// TwinCAT 3 PLC project DemoApplication
// ProgramVersion: 3.1.4020.4
// libraries:
//   Tc2_PfwLib_Processing, * (Beckhoff Automation GmbH)
//   Tc2_Standard, * (Beckhoff Automation GmbH)
//   Tc2_System, * (Beckhoff Automation GmbH)
//   Tc2_Utilities, * (Beckhoff Automation GmbH)
//   Tc3_Interfaces, * (Beckhoff Automation GmbH)
//   Tc3_Module, * (Beckhoff Automation GmbH)
//   VisuDialogs, * (System)
// project tree:
//   DUTs/ E_HMIstatus.TcDUT, E_MainStateMachine.TcDUT, ST_TempLoad.TcDUT, ST_TempLoad_Cmd.TcDUT, ST_TempLoad_State.TcDUT, ST_TempSave.TcDUT, ST_TempSave_Cmd.TcDUT
//   GVLs/ GVL_10_Visu.TcGVL, GVL_20_Applikation.TcGVL, GVL_30_Scope.TcGVL
//   / PlcTask.TcTTO
//   POUs/ FB_Load.TcPOU, FB_MainVisu.TcPOU, FB_Save.TcPOU, MAIN.TcPOU
//   TextLists/ GlobalTextList.TcGTLO, TL_Params_BOOL.TcTLO, TL_Params_Enum.TcTLO, TL_Params_INT.TcTLO, TL_Mparams_LREAL.TcTLO, TL_TcPfw_ErrorId.TcTLO, TL_Pparmas.TcTLO, TL_Supply.TcTLO, TL_TctrlOutSelect.TcTLO, TL_TctrlPowerTerminal.TcTLO, TL_TempSensType.TcTLO, TL_TerminalType.TcTLO
//   VISUs/DUTs/ st_ParamsUnsave.TcDUT, ST_Param_Visu.TcDUT
//   VISUs/Pages/Load Save/ Visu_SaveLoad.TcVIS
//   VISUs/Pages/LoopTest/ Visu_LoopTest.TcVIS
//   VISUs/Pages/Machine/Parameter/ Param_BOOL.TcVIS, Param_DINT.TcVIS, Param_ENUM_PowerTerm.TcVIS, Param_ENUM_SelOut.TcVIS, Param_ENUM_SensType.TcVIS, Param_ENUM_TermType.TcVIS, Param_LREAL.TcVIS
//   VISUs/Pages/Machine/Subpage/ Visu_Mparam_Autotune.TcVIS, Visu_Mparam_Cool.TcVIS, Visu_Mparam_Extruder.TcVIS, Visu_Mparam_General.TcVIS, Visu_Mparam_Heat.TcVIS, Visu_Mparam_Supply.TcVIS, Visu_Mparam_Temperatur.TcVIS
//   VISUs/Pages/Machine/ Visu_MParam.TcVIS
//   VISUs/Pages/Product/ Param_LREAL_Pparam.TcVIS, Visu_PParam.TcVIS, Visu_PParam_Params.TcVIS
//   VISUs/Pages/Supply/ Param_LREAL_Supply.TcVIS, Visu_Supply.TcVIS, Visu_Supply_Params.TcVIS
//   VISUs/Pages/ Visu_Main.TcVIS
//   VISUs/POUs/ FB_Visu_Param.TcPOU, FB_Visu_Pparam.TcPOU, FB_Visu_Supply.TcPOU
//   VISUs/ VisualizationManager.TcVMO (not stored)
// real-time tasks:
//   TASK PlcTask: cycle T#1ms, priority 20, ADS port 350
//   TASK Task 3: cycle T#10ms, priority 1, ADS port 351
// I/O:
//   DEVICE Device 1 (EtherCAT) (disabled), AmsNetId 192.168.1.78.2.1
//     Term 1 (EK1100) [EK1100 EtherCAT Coupler (2A E-Bus)]
//       Term 2 (EL3314) [EL3314 4Ch. Ana. Input Thermocouple (TC)]
//       Term 3 (EL2889) [EL2889 16Ch. Dig. Output 24V, 0.5A, negative]
// variable links:
//   DemoApplication/DemoApplication Instance <-> Device 1 (EtherCAT)/Term 1 (EK1100)/Term 3 (EL2889)
//     PlcTask Outputs/.out_PfwTempCtrlOutput[1]/Htr_PwmPos <-> Channel 1/Output

CONFIGURATION DemoApplication
    RESOURCE PLC ON TwinCAT3
        TASK PlcTask(INTERVAL := T#1ms, PRIORITY := 20);
        PROGRAM MAIN WITH PlcTask : MAIN;
    END_RESOURCE
END_CONFIGURATION

// ---- DUTs/E_HMIstatus.TcDUT
TYPE E_HMIstatus :
(
	Off := 0,
	Standby,
	On,
	Autotune,
	IdleLoad
);
END_TYPE

// ---- DUTs/E_MainStateMachine.TcDUT
TYPE E_MainStateMachine :
(
	eMainSM_BasicInit := 0,
	eMainSM_TempInit,
	eMainSM_MParamLoad,
	eMainSM_PParamLoad,
	eMainSM_SupParamLoad,
	eMainSM_StartUp,
	eMainSM_Idle
);
END_TYPE

// ---- DUTs/ST_TempLoad.TcDUT
TYPE ST_TempLoad :
STRUCT
	stTempCmd: ST_TempLoad_Cmd;
	stTempState: ST_TempLoad_State;
END_STRUCT
END_TYPE

// ---- DUTs/ST_TempLoad_Cmd.TcDUT
TYPE ST_TempLoad_Cmd :
STRUCT
	bLoadPparams: BOOL;
	bLoadMparams: BOOL;
	bLoadSupplyParams: BOOL;
END_STRUCT
END_TYPE

// ---- DUTs/ST_TempLoad_State.TcDUT
TYPE ST_TempLoad_State :
STRUCT
	bPparamLoaded: BOOL;
	bMparamLoaded: BOOL;
	bPparamLoad: BOOL;
	bMparamLoad: BOOL;
	bSupplyParamsLoad: BOOL;
	bSupplyParamsLoaded: BOOL;
END_STRUCT
END_TYPE

// ---- DUTs/ST_TempSave.TcDUT
TYPE ST_TempSave :
STRUCT
	stTempCmd: ST_TempSave_Cmd;
END_STRUCT
END_TYPE

// ---- DUTs/ST_TempSave_Cmd.TcDUT
TYPE ST_TempSave_Cmd :
STRUCT
	bSavePparams: BOOL;
	bSaveMparams: BOOL;
	bSaveSupplyParams: BOOL;
END_STRUCT
END_TYPE

// ---- VISUs/DUTs/st_ParamsUnsave.TcDUT
TYPE st_ParamsUnsave :
STRUCT
	mParams:	ARRAY[cnPfwTempCtrlFirst..cnPfwTempCtrlLast] OF BOOL;
	pParams:	ARRAY[cnPfwTempCtrlFirst..cnPfwTempCtrlLast] OF BOOL;
	supply:		ARRAY[cnPfwAppSupplyFirst..cnPfwAppSupplyLast] OF BOOL;
END_STRUCT
END_TYPE

// ---- VISUs/DUTs/ST_Param_Visu.TcDUT
TYPE ST_Param_Visu :
STRUCT
	 nActiveParamList: INT:=0;
	 
	sInUse:				STRING;
	 
	 bBoolAktValue:		ARRAY[1..cnParamsArrayLast] OF BOOL;
	 bBoolNewValue:		ARRAY[1..cnParamsArrayLast] OF BOOL;
	 bBoolSetValue:		ARRAY[1..cnParamsArrayLast] OF BOOL;

	 fLrealAktValue:	ARRAY[1..cnParamsArrayLast] OF LREAL;
	 fLrealNewValue:	ARRAY[1..cnParamsArrayLast] OF LREAL;
	 bLrealSetValue:	ARRAY[1..cnParamsArrayLast] OF BOOL;
	 
	 nDintAktValue:		ARRAY[1..cnParamsArrayLast] OF DINT;
	 nDintNewValue:		ARRAY[1..cnParamsArrayLast] OF DINT;
	 bDintSetValue:		ARRAY[1..cnParamsArrayLast] OF BOOL;
	 
	 nEnumAktValue:		ARRAY[1..cnParamsArrayLast] OF DINT;
	 nEnumNewValue:		ARRAY[1..cnParamsArrayLast] OF DINT;
	 bEnumSetValue:		ARRAY[1..cnParamsArrayLast] OF BOOL;
	 	 
END_STRUCT
END_TYPE

// ---- GVLs/GVL_10_Visu.TcGVL
VAR_GLOBAL CONSTANT
	cnParamsArrayLast:				INT:=50;
END_VAR

VAR_GLOBAL
	nVisuCount: INT:=cnPfwTempCtrlFirst;
	nSupplyCnt:	INT:=cnPfwAppSupplyFirst;
	
	eStatus: E_HMIstatus:=Off;
	
	bVisuNext: BOOL;
	bVisuBefore: BOOL;
	
	bVisuAutotune: BOOL;
	bVisuIdleLoad: BOOL;
	bVisuIdleLoadAktiv: BOOL;
	
	bGlobalError: BOOL;
	
	bParamsInit: BOOL:=FALSE;
	
	sErrorText:	STRING;
	
	
	
	
	stMParam_Visu:	ST_Param_Visu;
	stPParam_Visu:	ST_Param_Visu;
	stSupply_Visu:	ST_Param_Visu;
	stParamsUnsave:	st_ParamsUnsave;
	

	GlobalOne:INT:=1;
		A:INT:=0;
END_VAR

// ---- GVLs/GVL_20_Applikation.TcGVL
VAR_GLOBAL

	stTempLoad: ST_TempLoad;
	stTempSave: ST_TempSave;
	
END_VAR

// ---- GVLs/GVL_30_Scope.TcGVL
VAR_GLOBAL
	Scope_TempCtrlVariables: FB_Scope_TempCtrlVariables;
END_VAR

// ---- POUs/MAIN.TcPOU
PROGRAM MAIN
VAR
	eState: E_MainStateMachine := eMainSM_BasicInit;
	nCount: INT := 0;
	fCycleTime: LREAL := 0.025;
	fbTempCtrl: FB_TempCtrlMainBody_TcPfw_TC3;
	fbVisu: FB_MainVisu;

	bEntry:	BOOL;
	fbSave: FB_Save;
	fbLoad: FB_Load;
END_VAR


CASE eState OF
	eMainSM_BasicInit:
		_01_BasicInit();
		bEntry:=TRUE;
		eState:=eMainSM_MParamLoad;
		
	eMainSM_TempInit:
		_02_ParamsInit();
		bParamsInit:=FALSE;
		eState:=eMainSM_Idle;
		
	eMainSM_MParamLoad:
		IF bEntry THEN
			bEntry:=FALSE;
			stTempLoad.stTempCmd.bLoadMparams:=TRUE;
		ELSE
			IF stTempLoad.stTempState.bMparamLoaded THEN
				eState:=eMainSM_PParamLoad;
				bEntry:=TRUE;
			END_IF
		END_IF

		
	eMainSM_PParamLoad:
		IF bEntry THEN
			bEntry:=FALSE;
			stTempLoad.stTempCmd.bLoadPparams:=TRUE;
		ELSE
			IF stTempLoad.stTempState.bPparamLoaded THEN
				eState:=eMainSM_SupParamLoad;
				bEntry:=TRUE;
			END_IF
		END_IF

		
	eMainSM_SupParamLoad:
		IF bEntry THEN
			bEntry:=FALSE;
			stTempLoad.stTempCmd.bLoadSupplyParams:=TRUE;
		ELSE
			IF stTempLoad.stTempState.bSupplyParamsLoaded THEN
				eState:=eMainSM_StartUp;
				bEntry:=TRUE;
			END_IF
		END_IF

		
	eMainSM_StartUp:
		bEntry:=FALSE;
		fbTempCtrl.ConfigEnable:=TRUE;
		(*
		fbTempCtrl.tCycle:=fCycleTime;
		*)
		fbTempCtrl.tCycle:=0.025;
		fbTempCtrl.Looptest_Enable:=FALSE;
		fbTempCtrl.Callback_Enable:=TRUE;
		fbTempCtrl.Simu_Enable:=TRUE;
		eState:=eMainSM_Idle;
	
	eMainSM_Idle:
		IF bParamsInit THEN
			eState:=eMainSM_TempInit;
		END_IF
		
END_CASE

fbTempCtrl(
	Looptest_Enable:= TRUE,
	Scope_TempCtrlVariables:=Scope_TempCtrlVariables);
	
fbVisu();

fbSave();
fbLoad();

ACTION _01_BasicInit:
// Get Cycle Time
IF(GETCURTASKINDEXEX()<=0)THEN
	fCycletime:=0.025;		(* don't know, just guessing *)
ELSE
	fCycletime:=UDINT_TO_LREAL(_TaskInfo[GETCURTASKINDEXEX()].cycleTime)/10000000.0;
END_IF

// Init Zone ID/Name
FOR nCount := cnPfwTempCtrlFirst TO cnPfwTempCtrlLast DO
	aaaPfwTempMparamFromHmi[nCount].ZoneId := nCount;				(* zone id	*)
	aaaPfwTempMparamFromHmi[nCount].ZoneName := CONCAT('Zone_', INT_TO_STRING(nCount));	(* zonen name	*)
END_FOR
END_ACTION

ACTION _02_ParamsInit:
(* initialize of the machine parameter*)
	FOR nCount := cnPfwTempCtrlFirst TO cnPfwTempCtrlLast DO
		aaaPfwTempMparamFromHmi[nCount].AbsoluteHigh:=300;											(* limiting value of absolut hight.	*)
		aaaPfwTempMparamFromHmi[nCount].AbsoluteLow:=100;											(* limiting value of absolut low.	*)
		aaaPfwTempMparamFromHmi[nCount].InUse:=TRUE;												(* Zone is in use	*)
		aaaPfwTempMparamFromHmi[nCount].Enable:=TRUE;
		aaaPfwTempMparamFromHmi[nCount].SensorType:=0;												(* simulation	*)
		aaaPfwTempMparamFromHmi[nCount].ExtruderId:=1;												(* simulation	*)
		aaaPfwTempMparamFromHmi[nCount].TempSensTerm:=0;											(* simulation	*)
		aaaPfwTempMparamFromHmi[nCount].ZoneId:=nCount;												(* zone id		*)
		aaaPfwTempMparamFromHmi[nCount].ZoneName:=CONCAT('Zone_', INT_TO_STRING(nCount));(* zone name	*)
		IF(aaaPfwTempMparamFromHmi[nCount].KpCool<0.1)THEN
			aaaPfwTempMparamFromHmi[nCount].KpCool:=0.1;													(* default Kp cooling	*)
		END_IF
		IF(aaaPfwTempMparamFromHmi[nCount].KpHeat<0.1)THEN
			aaaPfwTempMparamFromHmi[nCount].KpHeat:=0.2;													(* default Kp heating 	*)
		END_IF
(*		aaaPfwTempMparamFromHmi[nCount].SettlingTime:=5.0;											(* Settling Time	*)*)
//		aaaPfwTempMparamFromHmi[nCount].SupplyLoad_Cooler:=100; 									(* coolingpower	*)
		aaaPfwTempMparamFromHmi[nCount].SupplyLoad_Heater:=1200;	 								(* heatingpower	*)
		aaaPfwTempMparamFromHmi[nCount].TuneEnd:=80;													(* Tune End % of setpoint	*)
		aaaPfwTempMparamFromHmi[nCount].TuneKp:=1.2;													(* Kp Tuning	*)
		aaaPfwTempMparamFromHmi[nCount].TuneTd:=0.25;												(* Td Tuning	*)
		aaaPfwTempMparamFromHmi[nCount].TuneTn:=2;													(* Tn Tuning	*)
		aaaPfwTempMparamFromHmi[nCount].TuneTv:=0.5;													(* Tv Tuning	*)
		aaaPfwTempMparamFromHmi[nCount].TuneY:=100;													(* Y Tuning		*)
		aaaPfwTempMparamFromHmi[nCount].Ramping_Rate:=0.005;										(* ramping rate	*)
		aaaPfwTempMparamFromHmi[nCount].Ramping_Tolerance:= 10;									(*	ramping tolerance*)
		aaaPfwTempMparamFromHmi[nCount].OutputSel_H:=eTcPfwTcOut_PWM;							(*	Heating output signal	*)
		aaaPfwTempMparamFromHmi[nCount].OutputSel_C:=eTcPfwTcOut_NoSignal;							(*	cooling output signal	*)
		aaaPfwTempMparamFromHmi[nCount].UseCooling:=FALSE;											(* cooling on	*)
		aaaPfwTempMparamFromHmi[nCount].TuneCooling:=FALSE;											(* cooling on	*)
		aaaPfwTempMparamFromHmi[nCount].ExtruderCompEna:=FALSE;											(* extruder comp	*)
		aaaPfwTempMparamFromHmi[nCount].fc_Enable:=FALSE;											(* Zwangskuelung	*)
		aaaPfwTempMparamFromHmi[nCount].fc_OffTime:=600.0;											(* Zwangskuelung	*)
		aaaPfwTempMparamFromHmi[nCount].fc_OnTime:=10.0;											(* Zwangskuelung	*)

(*		aaaPfwTempMparamFromHmi[nCount].SupplyLoad_Tolerance:=20.0;											(* Supply Tolerance	*)*)

		aaaPfwTempMparamFromHmi[nCount].SupplyLoad_Tolerance:=0.0;											(* Supply Tolerance	*)

		aaaPfwTempMparamFromHmi[nCount].SupplyId:=1;
		aaaPfwTempMparamFromHmi[nCount].ModuleId:=1;
	END_FOR
	(* mapping of the zones to the module and supply lines	*)


	(* initialize of the product parameter*)
	FOR nCount := cnPfwTempCtrlFirst TO cnPfwTempCtrlLast DO
		aaaPfwTempPparamFromHmi[nCount].Setpoint:=180;
		aaaPfwTempPparamFromHmi[nCount].StandbySetpoint:=18;
		aaaPfwTempPparamFromHmi[nCount].Threshold_M:=-10;
		aaaPfwTempPparamFromHmi[nCount].Threshold_MM:=-15;
		aaaPfwTempPparamFromHmi[nCount].Threshold_P:=10;
		aaaPfwTempPparamFromHmi[nCount].Threshold_PP:=15;
		aaaPfwTempPparamFromHmi[nCount].Update:=TRUE;
	END_FOR

	(* initialize of the supply lines*)
	FOR nCount := cnPfwAppSupplyFirst TO cnPfwAppSupplyLast DO
		stPfwSupplyLineCfg[nCount].fPwmCycleTime:=1;
		stPfwSupplyLineCfg[nCount].fPwmMaxOnTime:=1.0;
		stPfwSupplyLineCfg[nCount].fPwmMinOnTime:=0.1;
		stPfwSupplyLineCfg[nCount].fPwmMaxRampLoad:=1;
		stPfwSupplyLineCfg[nCount].nPwmFactorC:=10;
	END_FOR
END_ACTION

END_PROGRAM

// ---- POUs/FB_MainVisu.TcPOU
FUNCTION_BLOCK FB_MainVisu
VAR
	bOldVisuNext: BOOL;
	ncount: INT;
	bAutotuneAllDone: BOOL;
	eOldState: E_HMIstatus;
	bEntry:		BOOL:=TRUE;
	
	nIdx:				INT;
	fbVisuMParam:		FB_Visu_Param;
	fbVisuPParam:		FB_Visu_PParam;
	fbVisuSupply:		FB_Visu_Supply;
	(*
	fbVisu_Mparam:		FB_Visu_Mparam;
	fbVisu_Pparam:		FB_Visu_Pparam;
	fbVisu_Supply:		FB_Visu_Supply;
	*)
END_VAR

//
//		All Zones
//

bEntry:=(eStatus<>eOldState);
eOldState:=eStatus;

CASE eStatus OF

	Off:
		IF bEntry THEN
			FOR ncount:=cnPfwTempCtrlFirst TO cnPfwTempCtrlLast DO
				aaaPfwTempMparamFromHmi[ncount].Enable:=FALSE;
				stPfwTempCtrl[nCount].Enable:=FALSE;
			END_FOR
			bEntry:=FALSE;
		END_IF
	
	Standby:
		IF bEntry THEN
			FOR ncount:=cnPfwTempCtrlFirst TO cnPfwTempCtrlLast DO
				IF aaaPfwTempToHmi[nCount].InUse THEN
					stPfwTempCtrl[nCount].SelSetpoint:=TRUE;
					aaaPfwTempMparamFromHmi[ncount].Enable:=TRUE;
					stPfwTempCtrl[nCount].Enable:=TRUE;
				END_IF
			END_FOR
			bEntry:=FALSE;
		END_IF
	
	On:
		IF bEntry THEN
			FOR ncount:=cnPfwTempCtrlFirst TO cnPfwTempCtrlLast DO
				IF aaaPfwTempToHmi[nCount].InUse THEN
					stPfwTempCtrl[nCount].SelSetpoint:=FALSE;
					aaaPfwTempMparamFromHmi[ncount].Enable:=TRUE;
					stPfwTempCtrl[nCount].Enable:=TRUE;
				END_IF
			END_FOR
			bEntry:=FALSE;
		END_IF
	
	Autotune:
		IF bEntry THEN
			FOR ncount:=cnPfwTempCtrlFirst TO cnPfwTempCtrlLast DO
				IF aaaPfwTempToHmi[nCount].InUse THEN
					stPfwTempCtrl[nCount].Enable:=TRUE;
					aaaPfwTempMparamFromHmi[ncount].Enable:=TRUE;
					aaaPfwTempMparamFromHmi[ncount].Autotune:=TRUE;
				END_IF
			END_FOR
		ELSE
			bAutotuneAllDone:=TRUE;
			FOR ncount:=cnPfwTempCtrlFirst TO cnPfwTempCtrlLast DO
				IF(aaaPfwTempToHmi[nCount].TuningDone OR aaaPfwTempToHmi[nCount].Error) THEN
					IF aaaPfwTempToHmi[nCount].InUse THEN
						stPfwTempCtrl[nCount].Enable:=FALSE;
						aaaPfwTempMparamFromHmi[ncount].Enable:=FALSE;
						aaaPfwTempMparamFromHmi[ncount].Autotune:=FALSE;
					END_IF
				ELSE
					bAutoTuneAllDone:=FALSE;
				END_IF
			END_FOR
			IF bAutotuneAllDone THEN
				eStatus:=Standby;
			END_IF
		END_IF
		
	IdleLoad:
		IF bEntry THEN
			FOR ncount:=cnPfwTempCtrlFirst TO cnPfwTempCtrlLast DO
				IF aaaPfwTempToHmi[ncount].Enable THEN
					aaaPfwTempMparamFromHmi[ncount].Ena_TuneIdleLoad:=TRUE;
				END_IF
			END_FOR
		ELSE
			FOR ncount:=cnPfwTempCtrlFirst TO cnPfwTempCtrlLast DO
				bVisuIdleLoadAktiv:=FALSE;
				IF(aaaPfwTempToHmi[ncount].IdleLoadActive)THEN
					bVisuIdleLoadAktiv:=TRUE;
				END_IF
			END_FOR
			IF NOT bVisuIdleLoadAktiv THEN
				eStatus:=On;
			END_IF
		END_IF
END_CASE



//
//		Selected Zone
//

// Select Zone
IF(bVisuNext)THEN
	nVisuCount:=MIN(nVisuCount+1,cnPfwTempCtrlLast);
	bVisuNext:=FALSE;
ELSIF(bVisuBefore)THEN
	nVisuCount:=MAX(nVisuCount-1,cnPfwTempCtrlFirst);
	bVisuBefore:=FALSE;
END_IF

IF(bVisuAutotune)THEN
	aaaPfwTempMparamFromHmi[nVisuCount].Autotune:=TRUE;
ELSIF bVisuIdleLoad THEN
	aaaPfwTempMparamFromHmi[nVisuCount].Ena_TuneIdleLoad:=TRUE;
END_IF



ErrorHandling();
fbVisuMParam(stMParam_Visu:=stMParam_Visu, stParamsUnsave:=stParamsUnsave);
fbVisuPParam(stPParam_Visu:=stPParam_Visu, stParamsUnsave:=stParamsUnsave);
fbVisuSupply(stSupply_Visu:=stSupply_Visu, stParamsUnsave:=stParamsUnsave);

ACTION ErrorHandling:
bGlobalError:=FALSE;
sErrorText:='No Error';
FOR ncount:=cnPfwTempCtrlFirst TO cnPfwTempCtrlLast DO
	IF aaaPfwTempToHmi[ncount].Error THEN
		IF sErrorText='No Error' THEN
			sErrorText:='Error in Zone ';
		ELSE
			sErrorText:=CONCAT(sErrorText, ', ');
		END_IF
		sErrorText:=CONCAT(sErrorText, INT_TO_STRING(ncount));
		bGlobalError:=TRUE;
	END_IF
END_FOR
END_ACTION

END_FUNCTION_BLOCK

// ---- VISUs/POUs/FB_Visu_Param.TcPOU
FUNCTION_BLOCK FB_Visu_Param
VAR_IN_OUT
	stMParam_Visu:	ST_Param_Visu;
	stParamsUnsave:st_ParamsUnsave;
END_VAR
VAR
	nIdx:INT;
END_VAR

IF aaaPfwTempMparamFromHmi[nVisuCount].InUse THEN
	stMParam_Visu.sInUse:='Is In Use';
ELSE
	stMParam_Visu.sInUse:='Not In Use'; 
END_IF




FOR nIdx:=1 TO cnParamsArrayLast BY 1 DO
	// Get
	stMParam_Visu.bBoolAktValue[nIdx]:=GetBOOL(nVisuCount, nIdx);
	stMParam_Visu.fLrealAktValue[nIdx]:=GetLreal(nVisuCount, nIdx);
	stMParam_Visu.nDintAktValue[nIdx]:=GetInt(nVisuCount, nIdx);
	stMParam_Visu.nEnumAktValue[nIdx]:=GetEnum(nVisuCount, nIdx);
	
	// Set
	IF stMParam_Visu.bBoolSetValue[nIdx] THEN
		stMParam_Visu.bBoolSetValue[nIdx]:=FALSE;
		SetBool(nVisuCount,nIdx);
	END_IF
	
	IF stMParam_Visu.bLrealSetValue[nIdx] THEN
		stMParam_Visu.bLrealSetValue[nIdx]:=FALSE;
		SetLreal(nVisuCount,nIdx, stMParam_Visu.fLrealNewValue[nidx]);
	END_IF
	
	
	IF stMParam_Visu.bDintSetValue[nIdx] THEN
		stMParam_Visu.bDintSetValue[nIdx]:=FALSE;
		SetInt(nVisuCount,nIdx,DINT_TO_INT(stMParam_Visu.nDintNewValue[nidx]));
	END_IF
	
	IF stMParam_Visu.bEnumSetValue[nIdx] THEN
		stMParam_Visu.bEnumSetValue[nIdx]:=FALSE;
		SetEnum(nVisuCount,nIdx,stMParam_Visu.nEnumNewValue[nidx]);
	END_IF
END_FOR

METHOD SetInt : INT
VAR_INPUT
	nZone:	INT;
	nIdx:	INT;
	nValue:	INT;
END_VAR
CASE nIdx OF 
1:
	aaaPfwTempMparamFromHmi[nZone].App_HmiType:=nValue;
2:
	aaaPfwTempMparamFromHmi[nZone].TermChannel:=nValue;
3:
	aaaPfwTempMparamFromHmi[nZone].ExtruderId:=nValue;
4:
	aaaPfwTempMparamFromHmi[nZone].ModuleId:=nValue;
5:
	aaaPfwTempMparamFromHmi[nZone].ZoneId:=nValue;
6:
	aaaPfwTempMparamFromHmi[nZone].SupplyId:=nValue;
7:
	aaaPfwTempMparamFromHmi[nZone].CJ_CompMode:=nValue;
8:
	aaaPfwTempMparamFromHmi[nZone].CJ_CompZone:=nValue;
9:
	aaaPfwTempMparamFromHmi[nZone].SensTermSwapIdx:=nValue;
10:
	aaaPfwTempMparamFromHmi[nZone].HeaterSwapIdx:=nValue;
11:
	aaaPfwTempMparamFromHmi[nZone].CoolerSwapIdx:=nValue;
12:
	aaaPfwTempMparamFromHmi[nZone].nPwmFactorC:=nValue;

ELSE
	;
END_CASE

stParamsUnsave.mParams[nZone]:=TRUE;
END_METHOD

METHOD SetEnum : DINT
VAR_INPUT
	nZone:	INT;
	nIdx:	INT;
	nValue:	DINT;
END_VAR
CASE nIdx OF 

1:
	aaaPfwTempMparamFromHmi[nZone].OutputSel_H:=DINT_TO_INT(nValue);
2:
	aaaPfwTempMparamFromHmi[nZone].OutputSel_C:=DINT_TO_INT(nValue);
3:
	aaaPfwTempMparamFromHmi[nZone].TempSensTerm:=DINT_TO_INT(nValue);
4:
	aaaPfwTempMparamFromHmi[nZone].SensorType:=DINT_TO_INT(nValue);
ELSE
;
END_CASE
	
stParamsUnsave.mParams[nZone]:=TRUE;
END_METHOD

METHOD GetEnum : DINT
VAR_INPUT
	nZone:	INT;
	nIdx:	INT;
END_VAR
CASE nIdx OF 

1:
	GetEnum:=aaaPfwTempMparamFromHmi[nZone].OutputSel_H;
2:
	GetEnum:=aaaPfwTempMparamFromHmi[nZone].OutputSel_C;
3:
	GetEnum:=aaaPfwTempMparamFromHmi[nZone].TempSensTerm;
4:
	GetEnum:=aaaPfwTempMparamFromHmi[nZone].SensorType;
ELSE
	GetEnum:=-1;
END_CASE
END_METHOD

METHOD GetLreal : LREAL
VAR_INPUT
	nZone:	INT;
	nIdx:	INT;
END_VAR
VAR
END_VAR
CASE nIdx OF 
1:
	GetLreal:=aaaPfwTempMparamFromHmi[nZone].AbsoluteHigh;
2:
	GetLreal:=aaaPfwTempMparamFromHmi[nZone].AbsoluteLow;
3:
	GetLreal:=aaaPfwTempMparamFromHmi[nZone].ExtruderComp;
4:
	GetLreal:=aaaPfwTempMparamFromHmi[nZone].KpCool;
5:
	GetLreal:=aaaPfwTempMparamFromHmi[nZone].KpHeat;
6:
	GetLreal:=aaaPfwTempMparamFromHmi[nZone].TdCool;
7:
	GetLreal:=aaaPfwTempMparamFromHmi[nZone].TdHeat;
8:
	GetLreal:=aaaPfwTempMparamFromHmi[nZone].TnCool;
9:
	GetLreal:=aaaPfwTempMparamFromHmi[nZone].TnHeat;
10:
	GetLreal:=aaaPfwTempMparamFromHmi[nZone].TvCool;
11:
	GetLreal:=aaaPfwTempMparamFromHmi[nZone].TvHeat;
12:
	GetLreal:=aaaPfwTempMparamFromHmi[nZone].Overshoot;
13:
	GetLreal:=aaaPfwTempMparamFromHmi[nZone].Tracking_Rate;
14:
	GetLreal:=aaaPfwTempMparamFromHmi[nZone].Tracking_Td;
15:
	GetLreal:=aaaPfwTempMparamFromHmi[nZone].Ramping_Rate;
16:
	GetLreal:=aaaPfwTempMparamFromHmi[nZone].Ramping_RateC;
17:
	GetLreal:=aaaPfwTempMparamFromHmi[nZone].Ramping_Tolerance;
18:
	GetLreal:=aaaPfwTempMparamFromHmi[nZone].dTmax;
19:
	GetLreal:=aaaPfwTempMparamFromHmi[nZone].SensorOffset;
20:
	GetLreal:=aaaPfwTempMparamFromHmi[nZone].SettlingTime;
21:
	GetLreal:=aaaPfwTempMparamFromHmi[nZone].SupplyLoad_Cooler;
22:
	GetLreal:=aaaPfwTempMparamFromHmi[nZone].SupplyLoad_Heater;
23:
	GetLreal:=aaaPfwTempMparamFromHmi[nZone].SupplyLoad_Tolerance;
24:
	GetLreal:=aaaPfwTempMparamFromHmi[nZone].TuneEnd;
25:
	GetLreal:=aaaPfwTempMparamFromHmi[nZone].TuneKp;
26:
	GetLreal:=aaaPfwTempMparamFromHmi[nZone].TuneTd;
27:
	GetLreal:=aaaPfwTempMparamFromHmi[nZone].TuneTn;
28:
	GetLreal:=aaaPfwTempMparamFromHmi[nZone].TuneTv;
29:
	GetLreal:=aaaPfwTempMparamFromHmi[nZone].TuneTrackingTd;
30:
	GetLreal:=aaaPfwTempMparamFromHmi[nZone].TuneY;
31:
	GetLreal:=aaaPfwTempMparamFromHmi[nZone].L_LoadIdle;
32:
	GetLreal:=aaaPfwTempMparamFromHmi[nZone].Weighting_C;
33:
	GetLreal:=aaaPfwTempMparamFromHmi[nZone].ErrorHeatingFactor;
34:
	GetLreal:=aaaPfwTempMparamFromHmi[nZone].fPwmStdMaxOnTime;
35:(*
	F_GetMParamLreal:=aaaPfwTempMparamFromHmi[nZone].fPwmMaxOnTime;
	*)
	GetLreal:=0.0;
36:
	GetLreal:=aaaPfwTempMparamFromHmi[nZone].fPwmMinOnTime;
37:
	GetLreal:=aaaPfwTempMparamFromHmi[nZone].fc_OnTime;
38:
	GetLreal:=aaaPfwTempMparamFromHmi[nZone].fc_OffTime;
39:
	GetLreal:=aaaPfwTempMparamFromHmi[nZone].ActTempGain;
40:
	GetLreal:=aaaPfwTempMparamFromHmi[nZone].ActTempOffset;
	
ELSE
	GetLreal:=0.0;
END_CASE
END_METHOD

METHOD SetLreal : LREAL
VAR_INPUT
	nZone:	INT;
	nIdx:	INT;
	fValue:	LREAL;
END_VAR
VAR
END_VAR
CASE nIdx OF 
1:
	aaaPfwTempMparamFromHmi[nZone].AbsoluteHigh:=fValue;
2:
	aaaPfwTempMparamFromHmi[nZone].AbsoluteLow:=fValue;
3:
	aaaPfwTempMparamFromHmi[nZone].ExtruderComp:=fValue;
4:
	aaaPfwTempMparamFromHmi[nZone].KpCool:=fValue;
5:
	aaaPfwTempMparamFromHmi[nZone].KpHeat:=fValue;
6:
	aaaPfwTempMparamFromHmi[nZone].TdCool:=fValue;
7:
	aaaPfwTempMparamFromHmi[nZone].TdHeat:=fValue;
8:
	aaaPfwTempMparamFromHmi[nZone].TnCool:=fValue;
9:
	aaaPfwTempMparamFromHmi[nZone].TnHeat:=fValue;
10:
	aaaPfwTempMparamFromHmi[nZone].TvCool:=fValue;
11:
	aaaPfwTempMparamFromHmi[nZone].TvHeat:=fValue;
12:
	aaaPfwTempMparamFromHmi[nZone].Overshoot:=fValue;
13:
	aaaPfwTempMparamFromHmi[nZone].Tracking_Rate:=fValue;
14:
	aaaPfwTempMparamFromHmi[nZone].Tracking_Td:=fValue;
15:
	aaaPfwTempMparamFromHmi[nZone].Ramping_Rate:=fValue;
16:
	aaaPfwTempMparamFromHmi[nZone].Ramping_RateC:=fValue;
17:
	aaaPfwTempMparamFromHmi[nZone].Ramping_Tolerance:=fValue;
18:
	aaaPfwTempMparamFromHmi[nZone].dTmax:=fValue;
19:
	aaaPfwTempMparamFromHmi[nZone].SensorOffset:=fValue;
20:
	aaaPfwTempMparamFromHmi[nZone].SettlingTime:=fValue;
21:
	aaaPfwTempMparamFromHmi[nZone].SupplyLoad_Cooler:=fValue;
22:
	aaaPfwTempMparamFromHmi[nZone].SupplyLoad_Heater:=fValue;
23:
	aaaPfwTempMparamFromHmi[nZone].SupplyLoad_Tolerance:=fValue;
24:
	aaaPfwTempMparamFromHmi[nZone].TuneEnd:=fValue;
25:
	aaaPfwTempMparamFromHmi[nZone].TuneKp:=fValue;
26:
	aaaPfwTempMparamFromHmi[nZone].TuneTd:=fValue;
27:
	aaaPfwTempMparamFromHmi[nZone].TuneTn:=fValue;
28:
	aaaPfwTempMparamFromHmi[nZone].TuneTv:=fValue;
29:
	aaaPfwTempMparamFromHmi[nZone].TuneTrackingTd:=fValue;
30:
	aaaPfwTempMparamFromHmi[nZone].TuneY:=fValue;
31:
	aaaPfwTempMparamFromHmi[nZone].L_LoadIdle:=fValue;
32:
	aaaPfwTempMparamFromHmi[nZone].Weighting_C:=fValue;
33:
	aaaPfwTempMparamFromHmi[nZone].ErrorHeatingFactor:=fValue;
34:
	aaaPfwTempMparamFromHmi[nZone].fPwmStdMaxOnTime:=fValue;
35:(*
	F_GetMParamLreal:=aaaPfwTempMparamFromHmi[nZone].fPwmMaxOnTime;
	*)
	;
36:
	aaaPfwTempMparamFromHmi[nZone].fPwmMinOnTime:=fValue;
37:
	aaaPfwTempMparamFromHmi[nZone].fc_OnTime:=fValue;
38:
	aaaPfwTempMparamFromHmi[nZone].fc_OffTime:=fValue;
39:
	aaaPfwTempMparamFromHmi[nZone].ActTempGain:=fValue;
40:
	aaaPfwTempMparamFromHmi[nZone].ActTempOffset:=fValue;
	
ELSE
	;
END_CASE

stParamsUnsave.mParams[nZone]:=TRUE;
END_METHOD

METHOD SetBool : BOOL
VAR_INPUT
	nZone:	INT;
	nIdx:	INT;
END_VAR
CASE nIdx OF 

1:
	aaaPfwTempMparamFromHmi[nZone].UseCooling:= NOT aaaPfwTempMparamFromHmi[nZone].UseCooling;
2:
	aaaPfwTempMparamFromHmi[nZone].ExtruderCompEna:= NOT aaaPfwTempMparamFromHmi[nZone].ExtruderCompEna;
3:
	aaaPfwTempMparamFromHmi[nZone].TuneCooling:= NOT aaaPfwTempMparamFromHmi[nZone].TuneCooling;
4:
	aaaPfwTempMparamFromHmi[nZone].Tune_IdleLoad:= NOT aaaPfwTempMparamFromHmi[nZone].Tune_IdleLoad;
5:
	aaaPfwTempMparamFromHmi[nZone].Autotune:= NOT aaaPfwTempMparamFromHmi[nZone].Autotune;
6:
	aaaPfwTempMparamFromHmi[nZone].Enable:= NOT aaaPfwTempMparamFromHmi[nZone].Enable;
7:
	aaaPfwTempMparamFromHmi[nZone].Update:= NOT aaaPfwTempMparamFromHmi[nZone].Update;
8:
	aaaPfwTempMparamFromHmi[nZone].EnaExtruderBlock:= NOT aaaPfwTempMparamFromHmi[nZone].EnaExtruderBlock;
9:
	aaaPfwTempMparamFromHmi[nZone].NoFanWhileTrackDown:= NOT aaaPfwTempMparamFromHmi[nZone].NoFanWhileTrackDown;
10:
	aaaPfwTempMparamFromHmi[nZone].Ena_TuneIdleLoad:= NOT aaaPfwTempMparamFromHmi[nZone].Ena_TuneIdleLoad;
11:
	aaaPfwTempMparamFromHmi[nZone].LooptestUpdate:= NOT aaaPfwTempMparamFromHmi[nZone].LooptestUpdate;
12:
	aaaPfwTempMparamFromHmi[nZone].EnableErrorHeating:= NOT aaaPfwTempMparamFromHmi[nZone].EnableErrorHeating;
13:
	aaaPfwTempMparamFromHmi[nZone].ReadBack:= NOT aaaPfwTempMparamFromHmi[nZone].ReadBack;
14:
	aaaPfwTempMparamFromHmi[nZone].TuneExtruderComp:= NOT aaaPfwTempMparamFromHmi[nZone].TuneExtruderComp;
15:
	aaaPfwTempMparamFromHmi[nZone].TuneHeaterLoad:= NOT aaaPfwTempMparamFromHmi[nZone].TuneHeaterLoad;
16:
	aaaPfwTempMparamFromHmi[nZone].OpenloopHeating:= NOT aaaPfwTempMparamFromHmi[nZone].OpenloopHeating;
17:
	aaaPfwTempMparamFromHmi[nZone].fc_Enable:= NOT aaaPfwTempMparamFromHmi[nZone].fc_Enable;
18:
	aaaPfwTempMparamFromHmi[nZone].HibernateI_Cool:= NOT aaaPfwTempMparamFromHmi[nZone].HibernateI_Cool;
19:
	aaaPfwTempMparamFromHmi[nZone].hibernateI_Heat:= NOT aaaPfwTempMparamFromHmi[nZone].hibernateI_Heat;
20:
	aaaPfwTempMparamFromHmi[nZone].bSavingParams:= NOT aaaPfwTempMparamFromHmi[nZone].bSavingParams;
21:
	aaaPfwTempMparamFromHmi[nZone].bLoadParams:= NOT aaaPfwTempMparamFromHmi[nZone].bLoadParams;

ELSE
	SetBool:=FALSE;
END_CASE

stParamsUnsave.mParams[nZone]:=TRUE;
END_METHOD

METHOD GetInt : INT
VAR_INPUT
	nZone:	INT;
	nIdx:	INT;	
END_VAR
CASE nIdx OF 
1:
	GetInt:=aaaPfwTempMparamFromHmi[nZone].App_HmiType;
2:
	GetInt:=aaaPfwTempMparamFromHmi[nZone].TermChannel;
3:
	GetInt:=aaaPfwTempMparamFromHmi[nZone].ExtruderId;
4:
	GetInt:=aaaPfwTempMparamFromHmi[nZone].ModuleId;
5:
	GetInt:=aaaPfwTempMparamFromHmi[nZone].ZoneId;
6:
	GetInt:=aaaPfwTempMparamFromHmi[nZone].SupplyId;
7:
	GetInt:=aaaPfwTempMparamFromHmi[nZone].CJ_CompMode;
8:
	GetInt:=aaaPfwTempMparamFromHmi[nZone].CJ_CompZone;
9:
	GetInt:=aaaPfwTempMparamFromHmi[nZone].SensTermSwapIdx;
10:
	GetInt:=aaaPfwTempMparamFromHmi[nZone].HeaterSwapIdx;
11:
	GetInt:=aaaPfwTempMparamFromHmi[nZone].CoolerSwapIdx;
12:
	GetInt:=aaaPfwTempMparamFromHmi[nZone].nPwmFactorC;

ELSE
	GetInt:=0;
END_CASE
END_METHOD

METHOD GetBool : BOOL
VAR_INPUT
	nZone:	INT;
	nIdx:	INT;	
END_VAR
CASE nIdx OF 

1:
	GetBool:=aaaPfwTempMparamFromHmi[nZone].UseCooling;
2:
	GetBool:=aaaPfwTempMparamFromHmi[nZone].ExtruderCompEna;
3:
	GetBool:=aaaPfwTempMparamFromHmi[nZone].TuneCooling;
4:
	GetBool:=aaaPfwTempMparamFromHmi[nZone].Tune_IdleLoad;
5:
	GetBool:=aaaPfwTempMparamFromHmi[nZone].Autotune;
6:
	GetBool:=aaaPfwTempMparamFromHmi[nZone].Enable;
7:
	GetBool:=aaaPfwTempMparamFromHmi[nZone].Update;
8:
	GetBool:=aaaPfwTempMparamFromHmi[nZone].EnaExtruderBlock;
9:
	GetBool:=aaaPfwTempMparamFromHmi[nZone].NoFanWhileTrackDown;
10:
	GetBool:=aaaPfwTempMparamFromHmi[nZone].Ena_TuneIdleLoad;
11:
	GetBool:=aaaPfwTempMparamFromHmi[nZone].LooptestUpdate;
12:
	GetBool:=aaaPfwTempMparamFromHmi[nZone].EnableErrorHeating;
13:
	GetBool:=aaaPfwTempMparamFromHmi[nZone].ReadBack;
14:
	GetBool:=aaaPfwTempMparamFromHmi[nZone].TuneExtruderComp;
15:
	GetBool:=aaaPfwTempMparamFromHmi[nZone].TuneHeaterLoad;
16:
	GetBool:=aaaPfwTempMparamFromHmi[nZone].OpenloopHeating;
17:
	GetBool:=aaaPfwTempMparamFromHmi[nZone].fc_Enable;
18:
	GetBool:=aaaPfwTempMparamFromHmi[nZone].HibernateI_Cool;
19:
	GetBool:=aaaPfwTempMparamFromHmi[nZone].hibernateI_Heat;
20:
	GetBool:=aaaPfwTempMparamFromHmi[nZone].bSavingParams;
21:
	GetBool:=aaaPfwTempMparamFromHmi[nZone].bLoadParams;

ELSE
	GetBool:=FALSE;
END_CASE
END_METHOD

END_FUNCTION_BLOCK

// ---- VISUs/POUs/FB_Visu_Pparam.TcPOU
FUNCTION_BLOCK FB_Visu_Pparam
VAR_IN_OUT
	stPParam_Visu:	ST_Param_Visu;
	stParamsUnsave:st_ParamsUnsave;
END_VAR
VAR
	nIdx:INT;
END_VAR

// LREAL


FOR nIdx:=1 TO cnParamsArrayLast BY 1 DO
	// Get
	stPParam_Visu.fLrealAktValue[nIdx]:=GetLreal(nVisuCount, nIdx);
	

	IF stPParam_Visu.bLrealSetValue[nIdx] THEN
		stPParam_Visu.bLrealSetValue[nIdx]:=FALSE;
		SetLreal(nVisuCount,nIdx, stPParam_Visu.fLrealNewValue[nidx]);
	END_IF
END_FOR

METHOD SetLreal : LREAL
VAR_INPUT
	nZone:	INT;
	nIdx:	INT;
	fValue:	LREAL;
END_VAR
VAR
END_VAR
CASE nIdx OF 
1:
	aaaPfwTempPparamFromHmi[nZone].Setpoint:=fValue;
2:
	aaaPfwTempPparamFromHmi[nZone].StandbySetpoint:=fValue;
3:
	aaaPfwTempPparamFromHmi[nZone].Setpoints[1]:=fValue;
4:
	aaaPfwTempPparamFromHmi[nZone].Setpoints[2]:=fValue;
5:
	aaaPfwTempPparamFromHmi[nZone].Setpoints[3]:=fValue;
6:
	aaaPfwTempPparamFromHmi[nZone].Setpoints[4]:=fValue;
7:
	aaaPfwTempPparamFromHmi[nZone].Setpoints[5]:=fValue;
8:
	aaaPfwTempPparamFromHmi[nZone].Threshold_PP:=fValue;
9:
	aaaPfwTempPparamFromHmi[nZone].Threshold_P:=fValue;
10:
	aaaPfwTempPparamFromHmi[nZone].Threshold_M:=fValue;
11:
	aaaPfwTempPparamFromHmi[nZone].Threshold_MM:=fValue;
12:
	aaaPfwTempPparamFromHmi[nZone].Openloop_Output:=fValue;
ELSE
	;
END_CASE

stParamsUnsave.pParams[nZone]:=TRUE;
END_METHOD

METHOD GetLreal : LREAL
VAR_INPUT
	nZone:	INT;
	nIdx:	INT;
END_VAR
VAR
END_VAR
CASE nIdx OF 
1:
	GetLreal:=aaaPfwTempPparamFromHmi[nZone].Setpoint;
2:
	GetLreal:=aaaPfwTempPparamFromHmi[nZone].StandbySetpoint;
3:
	GetLreal:=aaaPfwTempPparamFromHmi[nZone].Setpoints[1];
4:
	GetLreal:=aaaPfwTempPparamFromHmi[nZone].Setpoints[2];
5:
	GetLreal:=aaaPfwTempPparamFromHmi[nZone].Setpoints[3];
6:
	GetLreal:=aaaPfwTempPparamFromHmi[nZone].Setpoints[4];
7:
	GetLreal:=aaaPfwTempPparamFromHmi[nZone].Setpoints[5];
8:
	GetLreal:=aaaPfwTempPparamFromHmi[nZone].Threshold_PP;
9:
	GetLreal:=aaaPfwTempPparamFromHmi[nZone].Threshold_P;
10:
	GetLreal:=aaaPfwTempPparamFromHmi[nZone].Threshold_M;
11:
	GetLreal:=aaaPfwTempPparamFromHmi[nZone].Threshold_MM;
12:
	GetLreal:=aaaPfwTempPparamFromHmi[nZone].Openloop_Output;
	
ELSE
	GetLreal:=0.0;
END_CASE
END_METHOD

END_FUNCTION_BLOCK

// ---- VISUs/POUs/FB_Visu_Supply.TcPOU
FUNCTION_BLOCK FB_Visu_Supply
VAR_IN_OUT
	stSupply_Visu:	ST_Param_Visu;
	stParamsUnsave:st_ParamsUnsave;
END_VAR
VAR_OUTPUT
END_VAR
VAR
	nidx:		INT;
END_VAR



// LREAL
FOR nIdx:=1 TO cnParamsArrayLast BY 1 DO
	
	// Get
	stSupply_Visu.fLrealAktValue[nIdx]:=GetLreal(nVisuCount, nIdx);
	
	//Set
	IF stSupply_Visu.bLrealSetValue[nIdx] THEN
		stSupply_Visu.bLrealSetValue[nIdx]:=FALSE;
		SetLreal(nVisuCount,nIdx, stSupply_Visu.fLrealNewValue[nidx]);
	END_IF
	
END_FOR

METHOD GetLreal : LREAL
VAR_INPUT
	nZone:	INT;
	nIdx:	INT;
END_VAR
CASE nIdx OF 
1:
	GetLreal:=stPfwSupplyLineCfg[nSupplyCnt].fPwmCycleTime;
2:
	GetLreal:=stPfwSupplyLineCfg[nSupplyCnt].fPwmMinOnTime;
3:
	GetLreal:=stPfwSupplyLineCfg[nSupplyCnt].fPwmMaxOnTime;
4:
	GetLreal:=stPfwSupplyLineCfg[nSupplyCnt].fPwmMaxOnC;
5:
	GetLreal:=stPfwSupplyLineCfg[nSupplyCnt].fPwmMaxRampLoad;
6:
	GetLreal:=stPfwSupplyLineCfg[nSupplyCnt].fActSupplyLoad;
7:
	GetLreal:=stPfwSupplyLineCfg[nSupplyCnt].fActSupplyLoad;
8:
	GetLreal:=stPfwSupplyLineCfg[nSupplyCnt].fActSupplyCurrent;
9:
	GetLreal:=stPfwSupplyLineCfg[nSupplyCnt].fSupplyLoad;
10:
	GetLreal:=stPfwSupplyLineCfg[nSupplyCnt].fSupplyMatch;

	
ELSE
	GetLreal:=0.0;
END_CASE
END_METHOD

METHOD SetLreal : LREAL
VAR_INPUT
	nZone:	INT;
	nIdx:	INT;
	fValue:	LREAL;
END_VAR
CASE nIdx OF 
1:
	stPfwSupplyLineCfg[nSupplyCnt].fPwmCycleTime:=fValue;
2:
	stPfwSupplyLineCfg[nSupplyCnt].fPwmMinOnTime:=fValue;
3:
	stPfwSupplyLineCfg[nSupplyCnt].fPwmMaxOnTime:=fValue;
4:
	stPfwSupplyLineCfg[nSupplyCnt].fPwmMaxOnC:=fValue;
5:
	stPfwSupplyLineCfg[nSupplyCnt].fPwmMaxRampLoad:=fValue;
6:
	stPfwSupplyLineCfg[nSupplyCnt].fActSupplyLoad:=fValue;
7:
	stPfwSupplyLineCfg[nSupplyCnt].fActSupplyLoad:=fValue;
8:
	stPfwSupplyLineCfg[nSupplyCnt].fActSupplyCurrent:=fValue;
9:
	stPfwSupplyLineCfg[nSupplyCnt].fSupplyLoad:=fValue;
10:
	stPfwSupplyLineCfg[nSupplyCnt].fSupplyMatch:=fValue;

	
ELSE
	SetLreal:=0.0;
END_CASE

stParamsUnsave.supply[nSupplyCnt]:=TRUE;
END_METHOD

END_FUNCTION_BLOCK

// ---- POUs/FB_Save.TcPOU
FUNCTION_BLOCK FB_Save
VAR

	nCount:				INT;
	bSavePparamsOld:	BOOL;
	bSaveMparamsOld:	BOOL;
	bSaveSupplyOld:		BOOL;
	
(* Old Routine *)
(*
	nSaveTemp: INT := cnPfwTempCtrlFirst;
	fbSaveParams: FB_TempParamSave_TcPfw;
	fbSaveSupplyParams: FB_TempSupplyParamSave_TcPfw;
	*)
END_VAR

(* save product parameters *)
IF(stTempSave.stTempCmd.bSavePparams AND NOT bSavePparamsOld)  THEN
	FOR nCount:=cnPfwTempCtrlFirst TO cnPfwTempCtrlLast DO
		IF	aaaPfwTempPparamFromHmi[nCount].SaveDelay=-1 THEN
			aaaPfwTempPparamFromHmi[nCount].SaveDelay:=100_000;
		END_IF
	END_FOR
ELSIF(stTempSave.stTempCmd.bSavePparams AND  bSavePparamsOld)  THEN
	stTempSave.stTempCmd.bSavePparams:=FALSE;
	FOR nCount:=cnPfwTempCtrlFirst TO cnPfwTempCtrlLast DO
		IF	aaaPfwTempPparamFromHmi[nCount].SaveDelay>-1 THEN
			stTempSave.stTempCmd.bSavePparams:=TRUE;
		END_IF
	END_FOR
END_IF
bSavePparamsOld:=stTempSave.stTempCmd.bSavePparams;


(* save machine parameters *)
IF(stTempSave.stTempCmd.bSaveMparams AND NOT bSaveMparamsOld)  THEN
	FOR nCount:=cnPfwTempCtrlFirst TO cnPfwTempCtrlLast DO
		IF	aaaPfwTempMparamFromHmi[nCount].SaveDelay=-1 THEN
			aaaPfwTempMparamFromHmi[nCount].SaveDelay:=100_000;
		END_IF
	END_FOR
ELSIF(stTempSave.stTempCmd.bSaveMparams AND  bSaveMparamsOld)  THEN
	stTempSave.stTempCmd.bSaveMparams:=FALSE;
	FOR nCount:=cnPfwTempCtrlFirst TO cnPfwTempCtrlLast DO
		IF	aaaPfwTempMparamFromHmi[nCount].SaveDelay>-1 THEN
			stTempSave.stTempCmd.bSaveMparams:=TRUE;
		END_IF
	END_FOR
	IF NOT stTempSave.stTempCmd.bSaveMparams THEN
		//bMParamUnsave:=FALSE;
		//MEMSET(ADR(bArMParamUnsave),0,SIZEOF(bArMParamUnsave));
	END_IF
END_IF
bSaveMparamsOld:=stTempSave.stTempCmd.bSaveMparams;


(* save supply lines *)
IF(stTempSave.stTempCmd.bSaveSupplyParams AND NOT bSaveSupplyOld)  THEN
	FOR nCount:=cnPfwAppSupplyFirst TO cnPfwAppSupplyLast DO
		IF	stPfwSupplyLineCfg[nCount].SaveDelay=-1 THEN
			stPfwSupplyLineCfg[nCount].SaveDelay:=100_000;
		END_IF
	END_FOR
ELSIF(stTempSave.stTempCmd.bSaveSupplyParams AND  bSaveSupplyOld)  THEN
	stTempSave.stTempCmd.bSaveSupplyParams:=FALSE;
	FOR nCount:=cnPfwAppSupplyFirst TO cnPfwAppSupplyLast DO
		IF	stPfwSupplyLineCfg[nCount].SaveDelay>-1 THEN
			stTempSave.stTempCmd.bSaveSupplyParams:=TRUE;
		END_IF
	END_FOR
END_IF
bSaveSupplyOld:=stTempSave.stTempCmd.bSaveSupplyParams;









(* Old Routine *)
(*

(* save product parameters *)
IF(stTempSave.stTempCmd.bSavePparams AND NOT stTempSave.stTempCmd.bSaveMparams AND NOT stTempSave.stTempCmd.bSaveSupplyParams)THEN
	IF(nSaveTemp>cnPfwTempCtrlLast)THEN
		nSaveTemp:=cnPfwTempCtrlFirst;
		stTempSave.stTempCmd.bSavePparams:=FALSE;
	ELSIF fbSaveParams.Execute AND (fbSaveParams.Done OR fbSaveParams.Error) THEN
		fbSaveParams.Execute:=FALSE;
		nSaveTemp:=nSaveTemp+1;
	ELSE
		fbSaveParams.PathName:=sPathP;
		fbSaveParams.Execute:=TRUE;
	END_IF
	fbSaveParams
		(
		Pparam:=aaaPfwTempPparamFromHmi[nSaveTemp],
		Mparam:=aaaPfwTempMparamFromHmi[nSaveTemp]
		);
END_IF

(* save supply lines *)
IF(stTempSave.stTempCmd.bSaveSupplyParams AND NOT stTempSave.stTempCmd.bSavePparams AND NOT stTempSave.stTempCmd.bSaveMparams)THEN
	IF(nSaveTemp>cnPfwAppSupplyLast)THEN
		nSaveTemp:=cnPfwAppSupplyFirst;
		stTempSave.stTempCmd.bSaveSupplyParams:=FALSE;
	ELSIF(fbSaveSupplyParams.Execute AND (fbSaveSupplyParams.Done OR fbSaveSupplyParams.Error))THEN
		fbSaveSupplyParams.Execute:=FALSE;
		nSaveTemp:=nSaveTemp+1;
	ELSE
		fbSaveSupplyParams.PathName:=sPathM;
		fbSaveSupplyParams.Execute:=TRUE;
	END_IF
	fbSaveSupplyParams
		(
		Supply:=stPfwSupplyLineCfg[nSaveTemp],
		supidx:=nSaveTemp
		);
END_IF

(* save machine parameters *)
IF(NOT stTempSave.stTempCmd.bSavePparams AND  stTempSave.stTempCmd.bSaveMparams AND NOT stTempSave.stTempCmd.bSaveSupplyParams)THEN
	IF(nSaveTemp>cnPfwTempCtrlLast)THEN
		nSaveTemp:=cnPfwTempCtrlFirst;
		stTempSave.stTempCmd.bSaveMparams:=FALSE;
	ELSIF(fbSaveParams.Execute AND (fbSaveParams.Done OR fbSaveParams.Error))THEN
		fbSaveParams.Execute:=FALSE;
		nSaveTemp:=nSaveTemp+1;
	ELSE
		fbSaveParams.PathName:=sPathM;
		fbSaveParams.Execute:=TRUE;
	END_IF
	fbSaveParams
		(
		Pparam:=aaaPfwTempPparamFromHmi[nSaveTemp],
		Mparam:=aaaPfwTempMparamFromHmi[nSaveTemp]
		);
END_IF

*)

END_FUNCTION_BLOCK

// ---- POUs/FB_Load.TcPOU
FUNCTION_BLOCK FB_Load
VAR
	
	nCount:				INT;
	
	(*
	Loadidx: INT;
	fbLoadParams: FB_TempParamLoad_TcPfw;
	fbLoadSupplyParams: FB_TempSupplyParamLoad_TcPfw;
	*)
END_VAR

(* product parameters *)
(* product parameter - Set load on true *)
IF (stTempLoad.stTempCmd.bLoadPparams AND NOT stTempLoad.stTempState.bPparamLoad) THEN
	stTempLoad.stTempCmd.bLoadPparams:=
	stTempLoad.stTempState.bPparamLoaded:=FALSE;
	stTempLoad.stTempState.bPparamLoad:=TRUE;
	FOR nCount:=cnPfwTempCtrlFirst TO cnPfwTempCtrlLast DO
		aaaPfwTempPparamFromHmi[nCount].bLoadParams:=TRUE;
	END_FOR
END_IF
(* product parameter - check load is done *)
IF stTempLoad.stTempState.bPparamLoad THEN
	stTempLoad.stTempState.bPparamLoad:=FALSE;
	FOR nCount:=cnPfwTempCtrlFirst TO cnPfwTempCtrlLast DO
		IF aaaPfwTempPparamFromHmi[nCount].bLoadParams THEN
			stTempLoad.stTempState.bPparamLoad:=TRUE;
		END_IF
	END_FOR
	stTempLoad.stTempState.bPparamLoaded:=NOT stTempLoad.stTempState.bPparamLoad;
END_IF



(* machine parameters *)
(* machine parameter - Set load on true *)
IF (stTempLoad.stTempCmd.bLoadMparams AND NOT stTempLoad.stTempState.bMparamLoad) THEN
	stTempLoad.stTempCmd.bLoadMparams:=
	stTempLoad.stTempState.bMparamLoaded:=FALSE;
	stTempLoad.stTempState.bMparamLoad:=TRUE;
	FOR nCount:=cnPfwTempCtrlFirst TO cnPfwTempCtrlLast DO
		aaaPfwTempMparamFromHmi[nCount].bLoadParams:=TRUE;
	END_FOR
END_IF
(* machine parameter - check load is done *)
IF stTempLoad.stTempState.bMparamLoad THEN
	stTempLoad.stTempState.bMparamLoad:=FALSE;
	FOR nCount:=cnPfwTempCtrlFirst TO cnPfwTempCtrlLast DO
		IF aaaPfwTempMparamFromHmi[nCount].bLoadParams THEN
			stTempLoad.stTempState.bPparamLoad:=TRUE;
		END_IF
	END_FOR
	stTempLoad.stTempState.bMparamLoaded:=NOT stTempLoad.stTempState.bMparamLoad;
END_IF



(* supply lines *)
(* supply lines - Set load on true *)
IF (stTempLoad.stTempCmd.bLoadSupplyParams AND NOT stTempLoad.stTempState.bSupplyParamsLoad) THEN
	stTempLoad.stTempCmd.bLoadSupplyParams:=
	stTempLoad.stTempState.bSupplyParamsLoaded:=FALSE;
	stTempLoad.stTempState.bSupplyParamsLoad:=TRUE;
	FOR nCount:=cnPfwAppSupplyFirst TO cnPfwAppSupplyLast DO
		stPfwSupplyLineCfg[nCount].bLoadParams:=TRUE;
	END_FOR
END_IF
(* supply lines - check load is done *)
IF stTempLoad.stTempState.bSupplyParamsLoad THEN
	stTempLoad.stTempState.bSupplyParamsLoad:=FALSE;
	FOR nCount:=cnPfwAppSupplyFirst TO cnPfwAppSupplyLast DO
		IF stPfwSupplyLineCfg[nCount].bLoadParams THEN
			stTempLoad.stTempState.bSupplyParamsLoad:=TRUE;
		END_IF
	END_FOR
	stTempLoad.stTempState.bSupplyParamsLoaded:=NOT stTempLoad.stTempState.bSupplyParamsLoad;
END_IF







(* Old Routine *)
(*
IF (stTempLoad.stTempCmd.bLoadPparams AND NOT stTempLoad.stTempCmd.bLoadMparams AND NOT stTempLoad.stTempCmd.bLoadSupplyParams)THEN
	IF(Loadidx<.cnPfwTempCtrlFirst)THEN
		stTempLoad.stTempState.bPparamLoaded:=FALSE;
		Loadidx:=cnPfwTempCtrlFirst;
		fbLoadParams.PathName:=sPathP;
	ELSIF(Loadidx>cnPfwTempCtrlLast)THEN
		Loadidx:=cnPfwTempCtrlFirst-1;
		stTempLoad.stTempState.bPparamLoaded:=TRUE;
		stTempLoad.stTempState.bPparamLoad:=FALSE;
		stTempLoad.stTempCmd.bLoadPparams:=FALSE;
	ELSE
		fbLoadParams
			(
			Mparam:=aaaPfwTempMparamFromHmi[Loadidx],
			Pparam:=aaaPfwTempPparamFromHmi[Loadidx],
			ProductParam:=TRUE
			);
		IF(fbLoadParams.Execute AND (fbLoadParams.Done OR fbLoadParams.Error))THEN
			fbLoadParams.Execute:=FALSE;
			Loadidx:=Loadidx+1;
		ELSE
			fbLoadParams.Execute:=TRUE;
		END_IF
	END_IF
END_IF

(*
load machine parameters 
*)
IF(NOT stTempLoad.stTempCmd.bLoadPparams AND  stTempLoad.stTempCmd.bLoadMparams AND NOT stTempLoad.stTempCmd.bLoadSupplyParams)THEN
	IF(Loadidx<cnPfwTempCtrlFirst)THEN
		stTempLoad.stTempState.bMparamLoaded:=FALSE;
		Loadidx:=cnPfwTempCtrlFirst;
		fbLoadParams.PathName:=sPathM;
	ELSIF(Loadidx>cnPfwTempCtrlLast)THEN
		Loadidx:=cnPfwTempCtrlFirst-1;
		stTempLoad.stTempState.bMparamLoaded:=TRUE;
		stTempLoad.stTempState.bMparamLoad:=FALSE;
		stTempLoad.stTempCmd.bLoadMparams:=FALSE;
	ELSE
		fbLoadParams
			(
			Mparam:=aaaPfwTempMparamFromHmi[Loadidx],
			Pparam:=aaaPfwTempPparamFromHmi[Loadidx],
			ProductParam:=FALSE
			);
		IF(fbLoadParams.Execute AND (fbLoadParams.Done OR fbLoadParams.Error))THEN
			fbLoadParams.Execute:=FALSE;
			Loadidx:=Loadidx+1;
		ELSE
			fbLoadParams.Execute:=TRUE;
		END_IF
	END_IF
END_IF

(*
load supply lines 
*)
IF(stTempLoad.stTempCmd.bLoadSupplyParams AND NOT stTempLoad.stTempCmd.bLoadPparams AND NOT stTempLoad.stTempCmd.bLoadMparams)THEN
	IF(Loadidx<cnPfwAppSupplyFirst)THEN
		stTempLoad.stTempState.bSupplyParamsLoaded:=FALSE;
		Loadidx:=cnPfwAppSupplyFirst;
		fbLoadSupplyParams.PathName:=sPathM;
	ELSIF(Loadidx>cnPfwAppSupplyLast)THEN
		Loadidx:=cnPfwTempCtrlFirst-1;
		stTempLoad.stTempState.bSupplyParamsLoaded:=TRUE;
		stTempLoad.stTempState.bSupplyParamsLoad:=FALSE;
		stTempLoad.stTempCmd.bLoadSupplyParams:=FALSE;
	ELSE
		fbLoadSupplyParams
			(
			Supply:=stPfwSupplyLineCfg[Loadidx],
			Supidx:=Loadidx
			);
		IF(fbLoadSupplyParams.Execute AND (fbLoadSupplyParams.Done OR fbLoadSupplyParams.Error))THEN
			fbLoadSupplyParams.Execute:=FALSE;
			Loadidx:=Loadidx+1;
		ELSE
			fbLoadSupplyParams.Execute:=TRUE;
		END_IF
	END_IF
END_IF
*)

END_FUNCTION_BLOCK

// ---- TextLists/GlobalTextList.TcGTLO
TEXTLIST GlobalTextList
  27 = '%5.2f'
  73 = '%5.3f'
  74 = '%5.4f'
  16 = '%d'
  33 = '%s'
  63 = '&s'
  66 = '+8'
  45 = '/s'
  9 = '632312'
  12 = '<'
  89 = '< previous Supply <'
  85 = '< previous Supply<'
  14 = '< previous Zone <'
  92 = '< Set <'
  91 = '<-'
  11 = '<<'
  69 = '<< -1 <<'
  71 = '<< -6 <<'
  70 = '<< -8 <<'
  94 = '<Set'
  93 = '<Set<'
  88 = '> next Supply >'
  87 = '> next Supply>'
  15 = '> next Zone >'
  68 = '>> +1 >>'
  72 = '>> +6 >>'
  67 = '>> +8 >>'
  30 = 'Actual Temperature'
  4 = 'All Zones'
  2 = 'Autotune'
  78 = 'BOOLs'
  18 = 'Commands'
  96 = 'Cool'
  29 = 'Cooling'
  79 = 'ENUMs'
  8 = 'Error'
  98 = 'Extruder'
  26 = 'f5.2'
  90 = 'General'
  7 = 'Global Reset'
  10 = 'GroupBox'
  95 = 'Heat'
  28 = 'Heating'
  3 = 'Idle Load'
  32 = 'IdleLoad'
  6 = 'Init Params'
  77 = 'INTs'
  65 = 'Is Unsave'
  38 = 'Load Machine'
  52 = 'Load Machineparameters'
  35 = 'Load Product'
  50 = 'Load Productparameters'
  40 = 'Load Supplylines'
  43 = 'Load Supplyparameters'
  58 = 'Loop Test'
  76 = 'LREALs'
  36 = 'Machine'
  47 = 'Main'
  55 = 'Maschine'
  53 = 'Maschine Params'
  60 = 'Maschinen Parameter'
  100 = 'Messurement Terminal'
  61 = 'Name:'
  62 = 'Not in Use'
  0 = 'Off'
  1 = 'On'
  5 = 'Operating State'
  17 = 'Parameter'
  31 = 'Power Level'
  13 = 'previous Zone'
  56 = 'Product'
  54 = 'Product Parameter'
  20 = 'rtData'
  48 = 'Save Load'
  37 = 'Save Machine'
  51 = 'Save Machineparameters'
  34 = 'Save Product'
  49 = 'Save Productparameters'
  39 = 'Save Supplylines'
  41 = 'Save SupplyParameters'
  42 = 'Save Supplyparameters'
  44 = 'Save/Load'
  86 = 'Selected Supply'
  46 = 'Selected Zone'
  75 = 'Set'
  19 = 'Setpoint'
  21 = 'Standby'
  57 = 'Supply'
  59 = 'Supply Parameter'
  84 = 'Switch'
  97 = 'Temperatur'
  80 = 'TEST'
  81 = 'TEST BOOL'
  83 = 'TEST ENUM'
  82 = 'TEST INT'
  22 = 'Thershold ++'
  23 = 'Threshold +'
  24 = 'Threshold -'
  25 = 'Threshold --'
  64 = 'Unsave'
  99 = 'Zone'
END_TEXTLIST

// ---- TextLists/TL_Params_BOOL.TcTLO
TEXTLIST TL_Params_BOOL
  1 = 'UseCooling' | en: 'a' | de: 'a'
  2 = 'ExtruderCompEna'
  3 = 'TuneCooling'
  4 = 'Tune_IdleLoad'
  5 = 'Autotune'
  6 = 'Enable'
  7 = 'Update'
  8 = 'EnaExtruderBlock'
  9 = 'NoFanWhileTrackDown'
  10 = 'Ena_TuneIdleLoad'
  11 = 'LooptestUpdate'
  12 = 'EnableErrorHeating'
  13 = 'ReadBack'
  14 = 'TuneExtruderComp'
  15 = 'TuneHeaterLoad'
  16 = 'OpenloopHeating'
  17 = 'fc_Enable'
  18 = 'HibernateI_Cool'
  19 = 'hibernateI_Heat'
  20 = 'bSavingParams'
  21 = 'bLoadParams'
  22 = '*** not Used ***'
  23 = '*** not Used ***'
  24 = '*** not Used ***'
  25 = '*** not Used ***'
  26 = '*** not Used ***'
  27 = '*** not Used ***'
  28 = '*** not Used ***'
  29 = '*** not Used ***'
  30 = '*** not Used ***'
  31 = '*** not Used ***'
  32 = '*** not Used ***'
  33 = '*** not Used ***'
  34 = '*** not Used ***'
  35 = '*** not Used ***'
  36 = '*** not Used ***'
  37 = '*** not Used ***'
  38 = '*** not Used ***'
  39 = '*** not Used ***'
  40 = '*** not Used ***'
   = ''
END_TEXTLIST

// ---- TextLists/TL_Params_Enum.TcTLO
TEXTLIST TL_Params_Enum
  1 = 'OutputSel_H'
  2 = 'OutputSel_C'
  3 = 'TempSensTerm'
  4 = 'SensorType'
  5 = '*** not Used ***'
  6 = '*** not Used ***'
  7 = '*** not Used ***'
  8 = '*** not Used ***'
  9 = '*** not Used ***'
   = ''
END_TEXTLIST

// ---- TextLists/TL_Params_INT.TcTLO
TEXTLIST TL_Params_INT
  1 = 'App_HmiType'
  2 = 'TermChannel'
  3 = 'ExtruderId'
  4 = 'ModuleId'
  5 = 'ZoneId'
  6 = 'SupplyId'
  7 = 'CJ_CompMode'
  8 = 'CJ_CompZone'
  9 = 'SensTermSwapIdx'
  10 = 'HeaterSwapIdx'
  11 = 'CoolerSwapIdx'
  12 = 'nPwmFactorC'
  13 = '*** not Used ***'
  14 = '*** not Used ***'
  15 = '*** not Used ***'
  16 = '*** not Used ***'
  17 = '*** not Used ***'
  18 = '*** not Used ***'
  19 = '*** not Used ***'
  20 = '*** not Used ***'
  21 = '*** not Used ***'
  22 = '*** not Used ***'
  23 = '*** not Used ***'
  24 = '*** not Used ***'
  25 = '*** not Used ***'
  26 = '*** not Used ***'
  27 = '*** not Used ***'
  28 = '*** not Used ***'
  29 = '*** not Used ***'
  30 = '*** not Used ***'
  31 = '*** not Used ***'
  32 = '*** not Used ***'
  33 = '*** not Used ***'
  34 = '*** not Used ***'
  35 = '*** not Used ***'
  36 = '*** not Used ***'
  37 = '*** not Used ***'
  38 = '*** not Used ***'
  39 = '*** not Used ***'
  40 = '*** not Used ***'
   = ''
END_TEXTLIST

// ---- TextLists/TL_Mparams_LREAL.TcTLO
TEXTLIST TL_Mparams_LREAL
  1 = 'AbsoluteHigh'
  2 = 'AbsoluteLow'
  3 = 'ExtruderComp'
  4 = 'KpCool'
  5 = 'KpHeat'
  6 = 'TdCool'
  7 = 'TdHeat'
  8 = 'TnCool'
  9 = 'TnHeat'
  10 = 'TvCool'
  11 = 'TvHeat'
  12 = 'Overshoot'
  13 = 'Tracking_Rate'
  14 = 'Tracking_Td'
  15 = 'Ramping_Rate'
  16 = 'Ramping_RateC'
  17 = 'Ramping_Tolerance'
  18 = 'dTmax'
  19 = 'SensorOffset'
  20 = 'SettlingTime'
  21 = 'SupplyLoad_Cooler'
  22 = 'SupplyLoad_Heater'
  23 = 'SupplyLoad_Tolerance'
  24 = 'TuneEnd'
  25 = 'TuneKp'
  26 = 'TuneTd'
  27 = 'TuneTn'
  28 = 'TuneTv'
  29 = 'TuneTrackingTd'
  30 = 'TuneY'
  31 = 'L_LoadIdle'
  32 = 'Weighting_C'
  33 = 'ErrorHeatingFactor'
  34 = 'fPwmStdMaxOnTime'
  35 = '*** not Used ***'
  36 = 'fPwmMinOnTime'
  37 = 'fc_OnTime'
  38 = 'fc_OffTime'
  39 = 'ActTempGain'
  40 = 'ActTempOffset'
  41 = 'SaveDelay'
   = ''
END_TEXTLIST

// ---- TextLists/TL_TcPfw_ErrorId.TcTLO
TEXTLIST TL_TcPfw_ErrorId
  0 = 'dwTcPfwTempErrNoError'
  4098 = 'dwTcPfwTempErrBusy'
  4099 = 'dwTcPfwTempTuneErr_NoTravel'
  4100 = 'dwTcPfwTempTuneErr_NoSettling'
  4101 = 'dwTcPfwTempTuneErr_Aborted'
  4102 = 'dwTcPfwTempTuneErr_ShortOfPoints'
  4103 = 'dwTcPfwTempTuneErr_NoTop'
  4104 = ''
  4105 = 'dwTcPfwTempTuneErr_NoResponse'
  17508 = 'dwTcPfwTempErrSnsHdwFailed'
  20464 = 'dwTcPfwTempErrDisconected'
  20465 = 'dwTcPfwTempErr_NoResponse'
  20466 = 'dwTcPfwTempErrNotOperational\n'
  20467 = 'dwTcPfwTempErrIoSwapCollision\n'
  20468 = 'dwTcPfwTempErrAdsSwapCollision\n'
  20469 = 'dwTcPfwTempErrInheritedFault\n'
  20478 = 'dwTcPfwTempErrOverCurrent\n'
  20479 = 'dwTcPfwTempErrUnderCurrent'
  20480 = 'dwTcPfwTempErrSnsCommFailed'
  1800 = 'dwTcPfwTempErrBusy'
  17489 = 'dwTcPfwTempErrSnsOverrun\n'
   = ''
END_TEXTLIST

// ---- TextLists/TL_Pparmas.TcTLO
TEXTLIST TL_Pparmas
  1 = 'Setpoint'
  2 = 'StandbySetpoint'
  3 = 'Setpoints[1]'
  4 = 'Setpoints[2]'
  5 = 'Setpoints[3]'
  6 = 'Setpoints[4]'
  7 = 'Setpoints[5]'
  8 = 'Threshold_PP'
  9 = 'Threshold_P'
  10 = 'Threshold_M'
  11 = 'Threshold_MM'
  12 = 'Openloop_Output'
   = ''
END_TEXTLIST

// ---- TextLists/TL_Supply.TcTLO
TEXTLIST TL_Supply
  1 = 'fPwmCycleTime'
  2 = 'fPwmMinOnTime'
  3 = 'fPwmMaxOnTime'
  4 = 'fPwmMaxOnC'
  5 = 'fPwmMaxRampLoad'
  6 = 'fActSupplyLoad'
  7 = 'fActSupplyLoad'
  8 = 'fActSupplyCurrent'
  9 = 'fSupplyLoad'
  10 = 'fSupplyMatch'
   = ''
END_TEXTLIST

// ---- TextLists/TL_TctrlOutSelect.TcTLO
TEXTLIST TL_TctrlOutSelect
  0 = 'NoSignal'
  1 = 'PWM'
  2 = 'Sign'
  3 = '2step'
   = ''
END_TEXTLIST

// ---- TextLists/TL_TctrlPowerTerminal.TcTLO
TEXTLIST TL_TctrlPowerTerminal
  0 = 'NoTerminal'
  1 = 'KL3403'
  2 = 'EL3403'
  3 = 'EL3773'
  4 = 'EL3x64'
  1000 = 'Simualtion'
  10000 = 'Customized'
   = ''
END_TEXTLIST

// ---- TextLists/TL_TempSensType.TcTLO
TEXTLIST TL_TempSensType
  0 = 'NoSensor'
  1 = 'TC_B'
  2 = 'TC_E'
  3 = 'TC_J'
  4 = 'TC_K'
  5 = 'TC_L'
  6 = 'TC_N'
  7 = 'TC_R'
  8 = 'TC_S'
  9 = 'TC_T'
  10 = 'TC_U'
  100 = 'PT_100'
  101 = 'NI_100'
  102 = 'NI_120'
  103 = 'PT_200'
  104 = 'PT_500'
  105 = 'PT_1000'
  106 = 'NI_1000'
  10000 = 'Customized'
   = ''
END_TEXTLIST

// ---- TextLists/TL_TerminalType.TcTLO
TEXTLIST TL_TerminalType
  0 = 'NoTerminal'
  1001 = 'KL300x'
  1002 = 'KL301x'
  1003 = 'KL302x'
  1004 = 'KL304x'
  1005 = 'KL305x'
  1006 = 'KL306x'
  1007 = 'KL310x'
  1008 = 'KL311x'
  1009 = 'KL312x'
  1010 = 'KL313x'
  1011 = 'KL314x'
  1012 = 'KL315x'
  1013 = 'KL317x'
  1014 = 'KL318x'
  1015 = 'KL340x'
  1016 = 'KL344x'
  1017 = 'KL346x'
  1018 = 'KL331x'
  2001 = 'EL331x'
  2002 = 'EL320x'
  2003 = 'EL316x'
  3001 = 'FM33xx'
  3002 = 'EM8908'
  10000 = 'Customized'
   = ''
END_TEXTLIST

// ---- VISUs/Pages/Load Save/Visu_SaveLoad.TcVIS
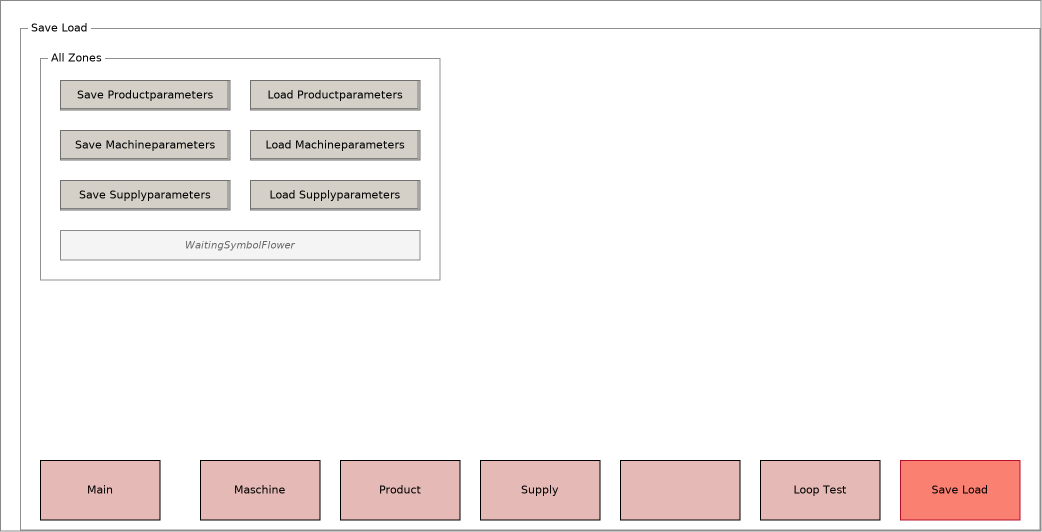
VISUALIZATION Visu_SaveLoad  // 1042x532
    GroupBox (20,20 1020x510), "Save Load"
        Rectangle (20,440 120x60), "Main"
            OnMouseClick: change screen: Visu_Main
        GroupBox (20,30 400x230), "All Zones", input disabled if: stTempSave.stTempCmd.bSaveMparams OR stTempSave.stTempCmd.bSaveSupplyParams OR stTempSave.stTempCmd.bSavePparams OR stTempLoad.stTempCmd.bLoadMparams OR stTempLoad.stTempCmd.bLoadPparams OR stTempLoad.stTempCmd.bLoadSupplyParams
            Button (20,30 170x30), "Save Productparameters"
                toggle stTempSave.stTempCmd.bSavePparams
            Button (210,30 170x30), "Load Productparameters"
                toggle stTempLoad.stTempCmd.bLoadPparams
            Button (20,80 170x30), "Save Machineparameters"
                toggle stTempSave.stTempCmd.bSaveMparams
            Button (210,80 170x30), "Load Machineparameters"
                toggle stTempLoad.stTempCmd.bLoadMparams
            Button (20,130 170x30), "Save Supplyparameters"
                toggle stTempSave.stTempCmd.bSaveSupplyParams
            Button (210,130 170x30), "Load Supplyparameters"
                toggle stTempLoad.stTempCmd.bLoadSupplyParams
            WaitingSymbolFlower (20,180 360x30), invisible if: NOT(stTempSave.stTempCmd.bSaveMparams OR stTempSave.stTempCmd.bSaveSupplyParams OR stTempSave.stTempCmd.bSavePparams OR stTempLoad.stTempCmd.bLoadMparams OR stTempLoad.stTempCmd.bLoadPparams OR stTempLoad.stTempCmd.bLoadSupplyParams)
        Rectangle (880,440 120x60), "Save Load"
            OnMouseClick: change screen: Visu_SaveLoad
        Rectangle (320,440 120x60), "Product"
            OnMouseClick: change screen: Visu_PParam
        Rectangle (180,440 120x60), "Maschine"
            OnMouseClick: change screen: Visu_MParam
        Rectangle (460,440 120x60), "Supply"
            OnMouseClick: change screen: Visu_Supply
        Rectangle (600,440 120x60)
        Rectangle (740,440 120x60), "Loop Test"
            OnMouseClick: change screen: Visu_LoopTest
END_VISUALIZATION

// ---- VISUs/Pages/LoopTest/Visu_LoopTest.TcVIS
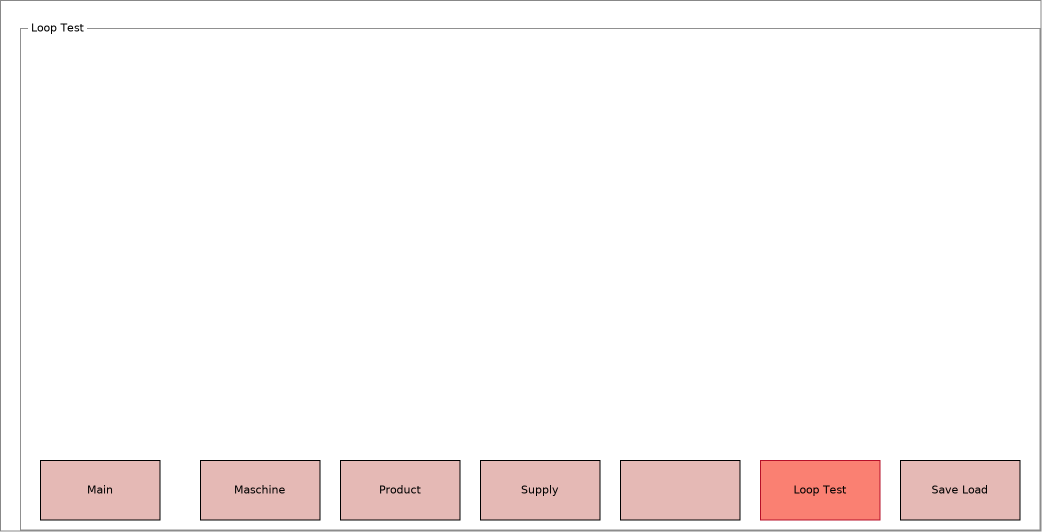
VISUALIZATION Visu_LoopTest  // 1042x532
    GroupBox (20,20 1020x510), "Loop Test"
        Rectangle (20,440 120x60), "Main"
            OnMouseClick: change screen: Visu_Main
        Rectangle (880,440 120x60), "Save Load"
            OnMouseClick: change screen: Visu_SaveLoad
        Rectangle (320,440 120x60), "Product"
            OnMouseClick: change screen: Visu_PParam
        Rectangle (180,440 120x60), "Maschine"
            OnMouseClick: change screen: Visu_MParam
        Rectangle (460,440 120x60), "Supply"
            OnMouseClick: change screen: Visu_Supply
        Rectangle (600,440 120x60)
        Rectangle (740,440 120x60), "Loop Test"
            OnMouseClick: change screen: Visu_LoopTest
END_VISUALIZATION

// ---- VISUs/Pages/Machine/Parameter/Param_BOOL.TcVIS
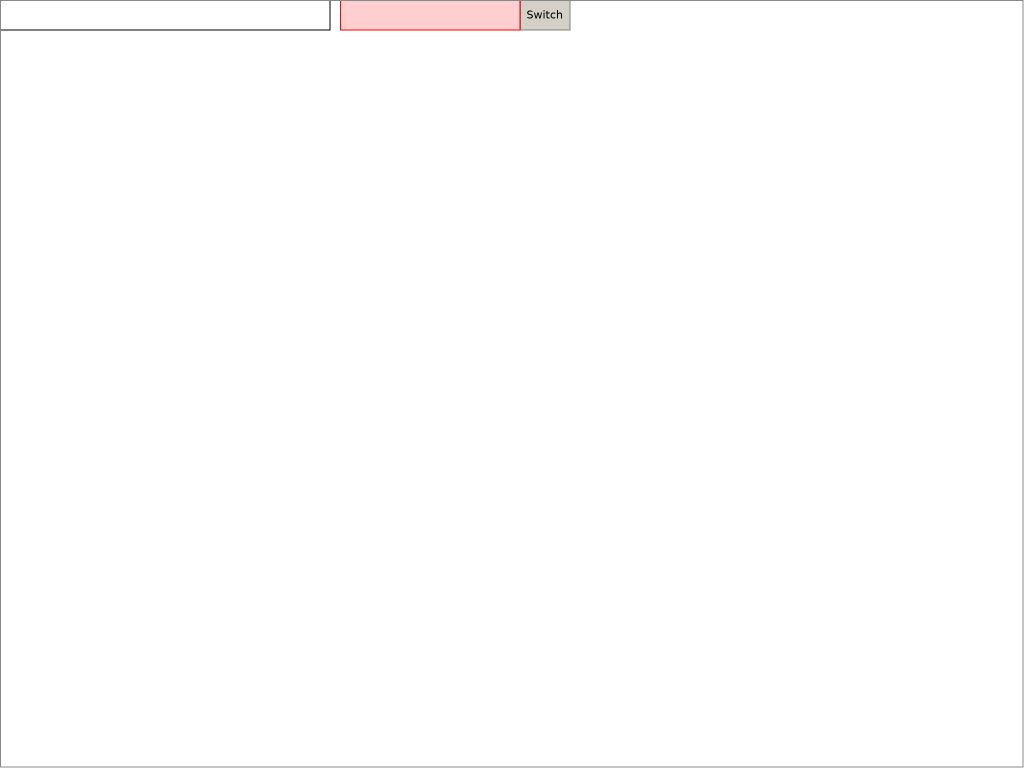
VISUALIZATION Param_BOOL  // 1024x768
VAR_INPUT
	nIdx:		INT;
END_VAR
    Rectangle (0,0 330x30), text list: 'TL_Params_BOOL', text index: nIdx
    Rectangle (520,0 50x30), "Switch", colour toggle: stMParam_Visu.bBoolSetValue[nIdx]
        OnMouseClick: execute { stMParam_Visu.bBoolSetValue[nIdx]:=TRUE; }
    Rectangle (340,0 180x30), colour toggle: stMParam_Visu.bBoolAktValue[nIdx]
    Rectangle (600,0 150x30)
END_VISUALIZATION

// ---- VISUs/Pages/Machine/Parameter/Param_DINT.TcVIS
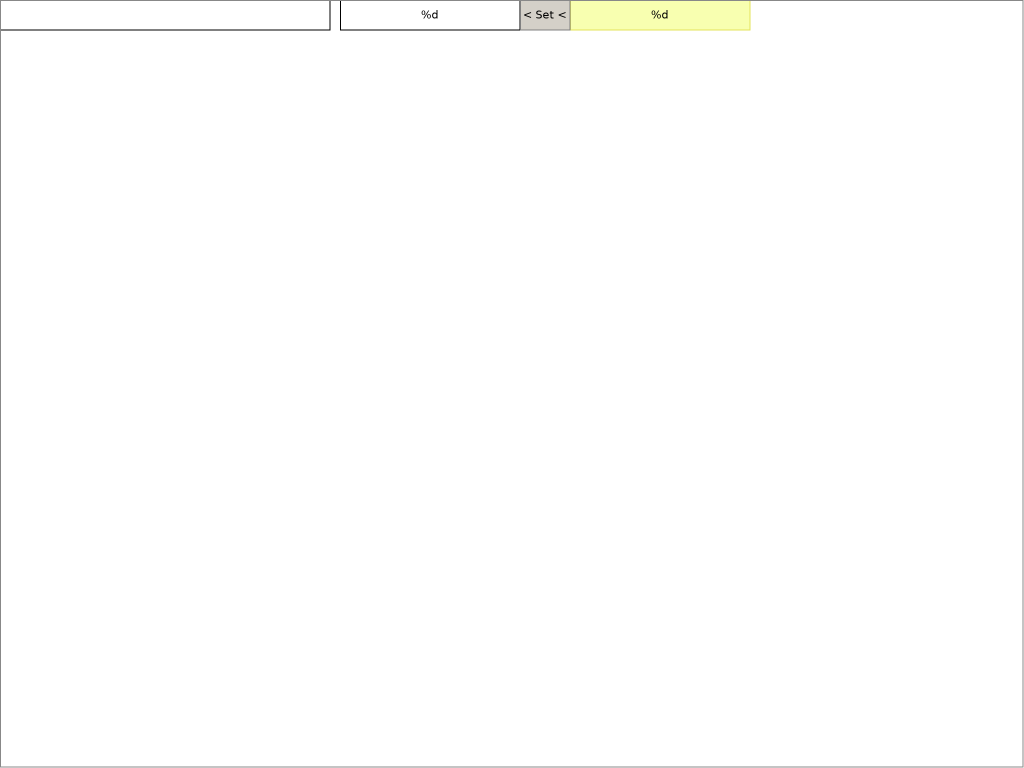
VISUALIZATION Param_DINT  // 1024x768
VAR_INPUT
	nIdx:		INT;
END_VAR
    Rectangle (340,0 180x30), "%d", text variable: stMParam_Visu.nDintAktValue[nIdx]
    Rectangle (0,0 330x30), text list: 'TL_Params_INT', text index: nIdx
    Rectangle (570,0 180x30), "%d", text variable: stMParam_Visu.nDintNewValue[nIdx]
        OnMouseClick: write the text variable via Default
    Rectangle (520,0 50x30), "< Set <"
        OnMouseClick: execute { stMParam_Visu.bDintSetValue[nIdx]:=TRUE; }
END_VISUALIZATION

// ---- VISUs/Pages/Machine/Parameter/Param_ENUM_PowerTerm.TcVIS
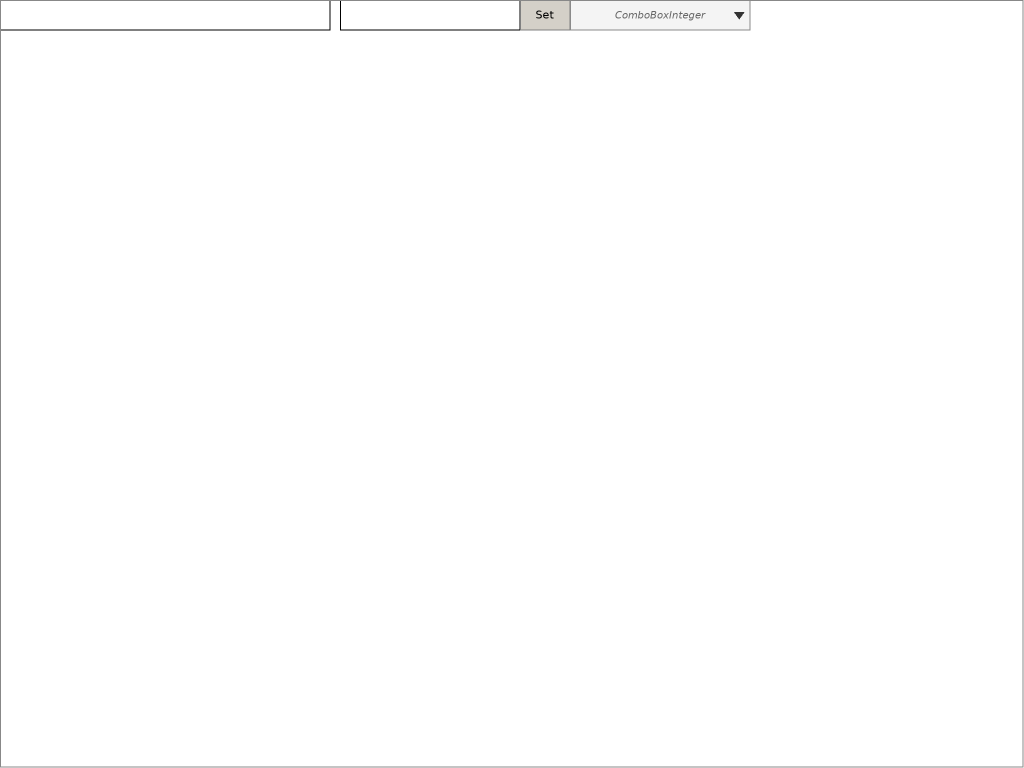
VISUALIZATION Param_ENUM_PowerTerm  // 1024x768
VAR_INPUT
	nIdx:		INT;
END_VAR
    Rectangle (340,0 180x30), text list: 'TL_TctrlPowerTerminal', text index: stMParam_Visu.nEnumAktValue[nIdx]
    Rectangle (0,0 330x30), text list: 'TL_Params_Enum', text index: nIdx
    Rectangle (520,0 50x30), "Set"
        OnMouseClick: execute { stMParam_Visu.bEnumSetValue[nIdx]:=TRUE; }
    ComboBoxInteger (570,0 180x30), variable: stMParam_Visu.nEnumNewValue[nIdx], text list: 'TL_TctrlPowerTerminal'
END_VISUALIZATION

// ---- VISUs/Pages/Machine/Parameter/Param_ENUM_SelOut.TcVIS
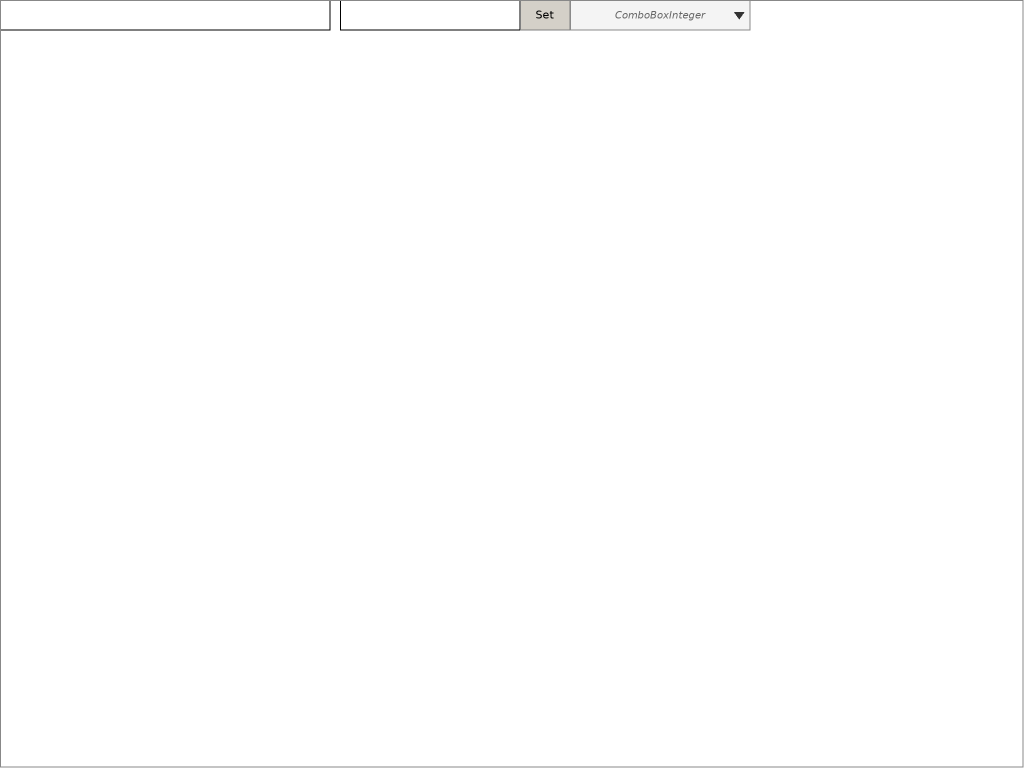
VISUALIZATION Param_ENUM_SelOut  // 1024x768
VAR_INPUT
	nIdx:		INT;
END_VAR
    Rectangle (340,0 180x30), text list: 'TL_TctrlOutSelect', text index: stMParam_Visu.nEnumAktValue[nIdx]
    Rectangle (0,0 330x30), text list: 'TL_Params_Enum', text index: nIdx
    Rectangle (520,0 50x30), "Set"
        OnMouseClick: execute { stMParam_Visu.bEnumSetValue[nIdx]:=TRUE; }
    ComboBoxInteger (570,0 180x30), variable: stMParam_Visu.nEnumNewValue[nIdx], text list: 'TL_TctrlOutSelect'
END_VISUALIZATION

// ---- VISUs/Pages/Machine/Parameter/Param_ENUM_SensType.TcVIS
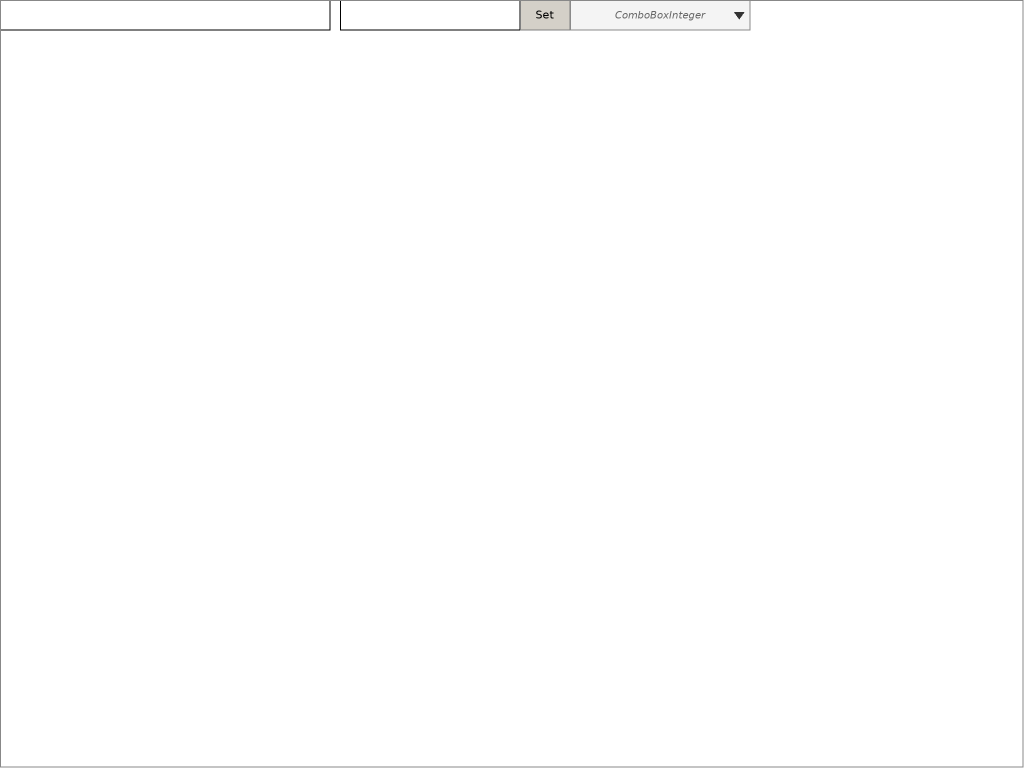
VISUALIZATION Param_ENUM_SensType  // 1024x768
VAR_INPUT
	nIdx:		INT;
END_VAR
    Rectangle (340,0 180x30), text list: 'TL_TempSensType', text index: stMParam_Visu.nEnumAktValue[nIdx]
    Rectangle (0,0 330x30), text list: 'TL_Params_Enum', text index: nIdx
    Rectangle (520,0 50x30), "Set"
        OnMouseClick: execute { stMParam_Visu.bEnumSetValue[nIdx]:=TRUE; }
    ComboBoxInteger (570,0 180x30), variable: stMParam_Visu.nEnumNewValue[nIdx], text list: 'TL_TempSensType'
END_VISUALIZATION

// ---- VISUs/Pages/Machine/Parameter/Param_ENUM_TermType.TcVIS
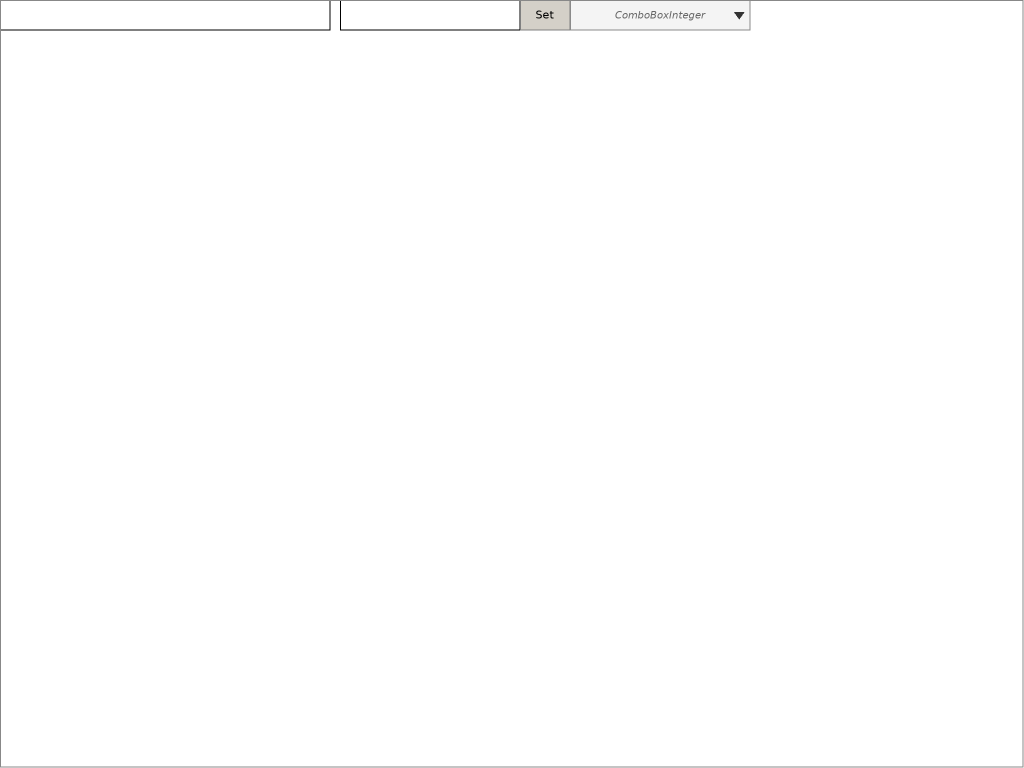
VISUALIZATION Param_ENUM_TermType  // 1024x768
VAR_INPUT
	nIdx:		INT;
END_VAR
    Rectangle (340,0 180x30), text list: 'TL_TerminalType', text index: stMParam_Visu.nEnumAktValue[nIdx]
    Rectangle (0,0 330x30), text list: 'TL_Params_Enum', text index: nIdx
    Rectangle (520,0 50x30), "Set"
        OnMouseClick: execute { stMParam_Visu.bEnumSetValue[nIdx]:=TRUE; }
    ComboBoxInteger (570,0 180x30), variable: stMParam_Visu.nEnumNewValue[nIdx], text list: 'TL_TerminalType'
END_VISUALIZATION

// ---- VISUs/Pages/Machine/Parameter/Param_LREAL.TcVIS
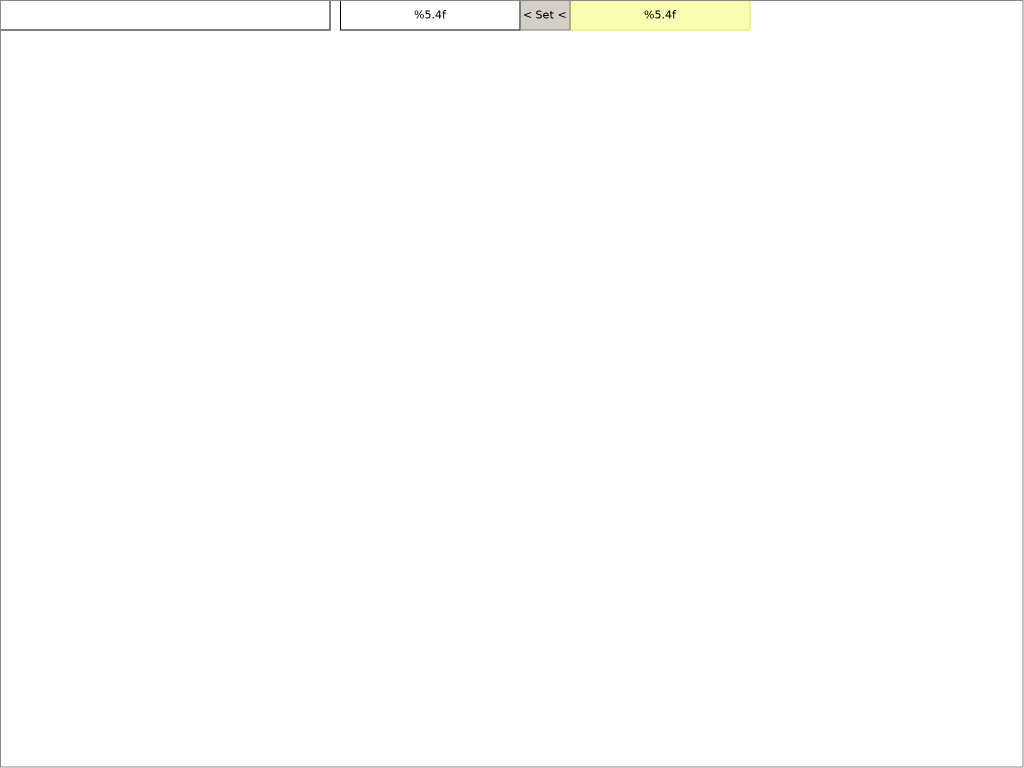
VISUALIZATION Param_LREAL  // 1024x768
VAR_INPUT
	nIdx:		INT;
END_VAR
    Rectangle (340,0 180x30), "%5.4f", text variable: stMParam_Visu.fLrealAktValue[nIdx]
    Rectangle (0,0 330x30), text list: 'TL_Mparams_LREAL', text index: nIdx
    Rectangle (570,0 180x30), "%5.4f", text variable: stMParam_Visu.fLrealNewValue[nIdx]
        OnMouseClick: write the text variable via Default
    Rectangle (520,0 50x30), "< Set <"
        OnMouseClick: execute { stMParam_Visu.bLrealSetValue[nIdx]:=TRUE; }
END_VISUALIZATION

// ---- VISUs/Pages/Machine/Subpage/Visu_Mparam_Autotune.TcVIS
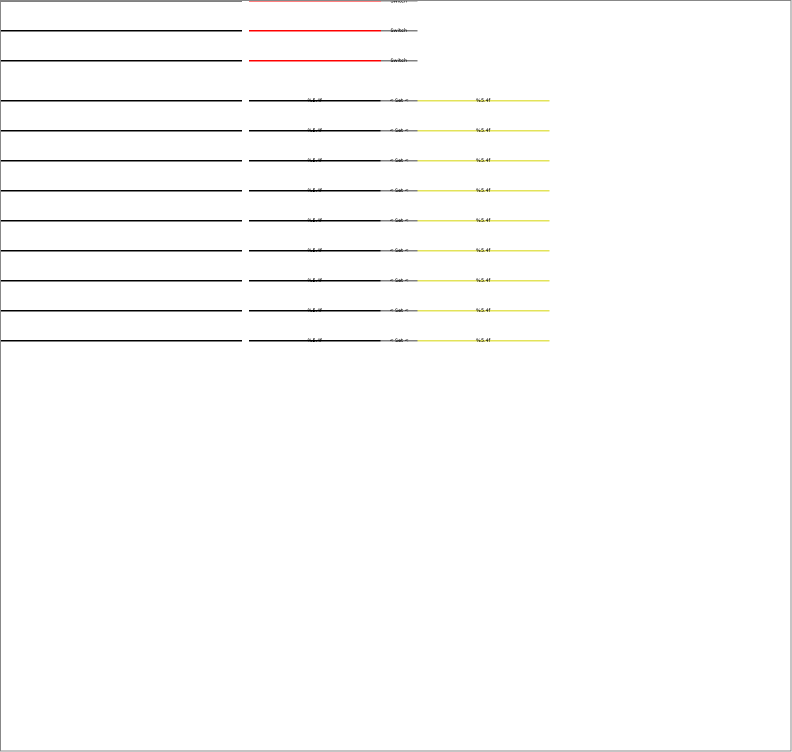
VISUALIZATION Visu_Mparam_Autotune  // 792x752
    Frame (0,100 750x30)
        shows Param_LREAL(nIdx := 24)
    Frame (0,130 750x30)
        shows Param_LREAL(nIdx := 25)
    Frame (0,160 750x30)
        shows Param_LREAL(nIdx := 26)
    Frame (0,190 750x30)
        shows Param_LREAL(nIdx := 27)
    Frame (0,220 750x30)
        shows Param_LREAL(nIdx := 28)
    Frame (0,250 750x30)
        shows Param_LREAL(nIdx := 29)
    Frame (0,280 750x30)
        shows Param_LREAL(nIdx := 30)
    Frame (0,310 750x30)
        shows Param_LREAL(nIdx := 31)
    Frame (0,340 750x30)
        shows Param_LREAL(nIdx := 23)
    Frame (0,60 750x30)
        shows Param_BOOL(nIdx := 10)
    Frame (0,30 750x30)
        shows Param_BOOL(nIdx := 4)
    Frame (0,0 750x30)
        shows Param_BOOL(nIdx := 5)
    Rectangle (40,720 750x30)
END_VISUALIZATION

// ---- VISUs/Pages/Machine/Subpage/Visu_Mparam_Cool.TcVIS
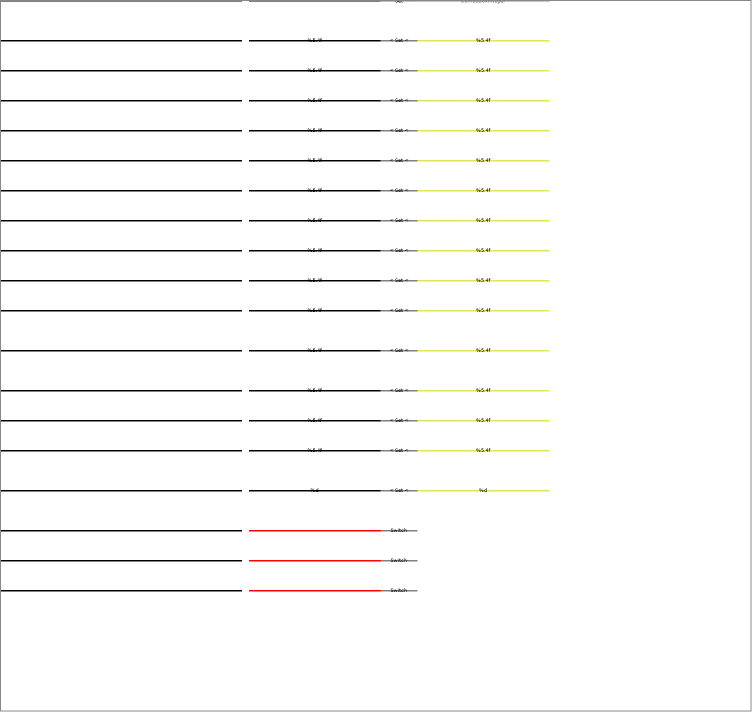
VISUALIZATION Visu_Mparam_Cool  // 752x712
    Frame (0,40 750x30)
        shows Param_LREAL(nIdx := 5)
    Frame (0,70 750x30)
        shows Param_LREAL(nIdx := 7)
    Frame (0,100 750x30)
        shows Param_LREAL(nIdx := 9)
    Frame (0,130 750x30)
        shows Param_LREAL(nIdx := 11)
    Frame (0,490 750x30)
        shows Param_DINT(nIdx := 10)
    Frame (0,0 750x30)
        shows Param_ENUM_SelOut(nIdx := 2)
    Frame (0,160 750x30)
        shows Param_LREAL(nIdx := 12)
    Frame (0,190 750x30)
        shows Param_LREAL(nIdx := 13)
    Frame (0,220 750x30)
        shows Param_LREAL(nIdx := 14)
    Frame (0,250 750x30)
        shows Param_LREAL(nIdx := 15)
    Frame (0,280 750x30)
        shows Param_LREAL(nIdx := 17)
    Frame (0,310 750x30)
        shows Param_LREAL(nIdx := 18)
    Frame (0,350 750x30)
        shows Param_LREAL(nIdx := 22)
    Frame (0,390 750x30)
        shows Param_LREAL(nIdx := 33)
    Frame (0,420 750x30)
        shows Param_LREAL(nIdx := 34)
    Frame (0,450 750x30)
        shows Param_LREAL(nIdx := 36)
    Frame (0,530 750x30)
        shows Param_BOOL(nIdx := 12)
    Frame (0,560 750x30)
        shows Param_BOOL(nIdx := 16)
    Frame (0,590 750x30)
        shows Param_BOOL(nIdx := 19)
    Rectangle (0,680 750x30)
END_VISUALIZATION

// ---- VISUs/Pages/Machine/Subpage/Visu_Mparam_Extruder.TcVIS
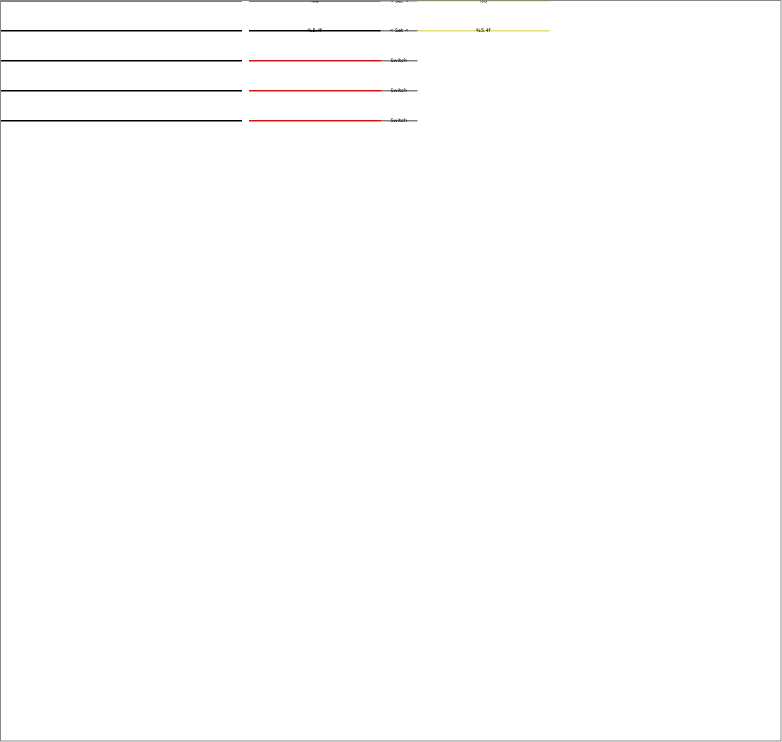
VISUALIZATION Visu_Mparam_Extruder  // 782x742
    Frame (0,30 750x30)
        shows Param_LREAL(nIdx := 3)
    Frame (0,90 750x30)
        shows Param_BOOL(nIdx := 8)
    Frame (0,60 750x30)
        shows Param_BOOL(nIdx := 2)
    Frame (0,0 750x30)
        shows Param_DINT(nIdx := 3)
    Frame (0,120 750x30)
        shows Param_BOOL(nIdx := 14)
    Rectangle (30,710 750x30)
END_VISUALIZATION

// ---- VISUs/Pages/Machine/Subpage/Visu_Mparam_General.TcVIS
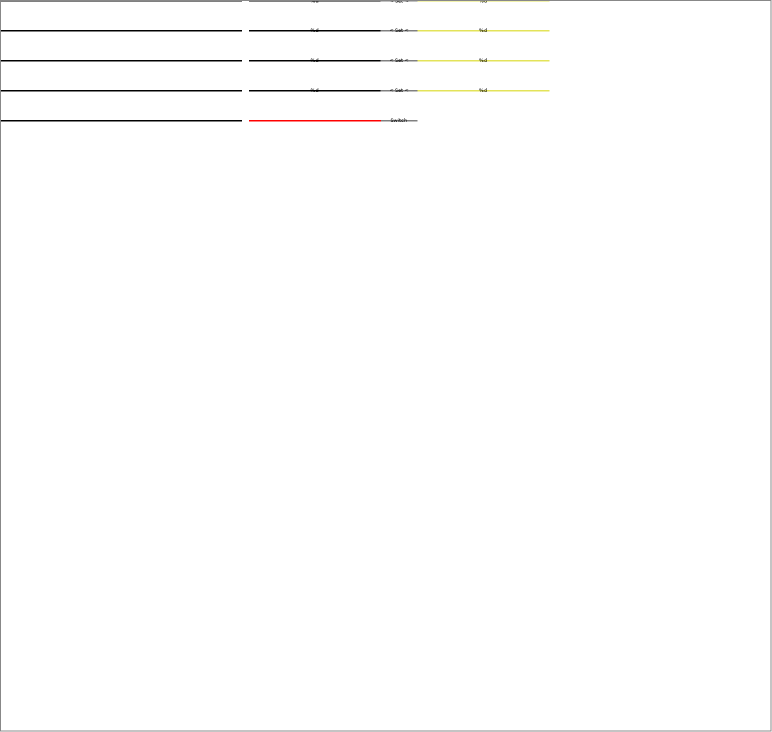
VISUALIZATION Visu_Mparam_General  // 772x732
    Frame (0,120 750x30)
        shows Param_BOOL(nIdx := 6)
    Frame (0,0 750x30)
        shows Param_DINT(nIdx := 3)
    Frame (0,30 750x30)
        shows Param_DINT(nIdx := 4)
    Frame (0,60 750x30)
        shows Param_DINT(nIdx := 5)
    Frame (0,90 750x30)
        shows Param_DINT(nIdx := 6)
    Rectangle (10,690 750x30)
    Rectangle (20,700 750x30)
END_VISUALIZATION

// ---- VISUs/Pages/Machine/Subpage/Visu_Mparam_Heat.TcVIS
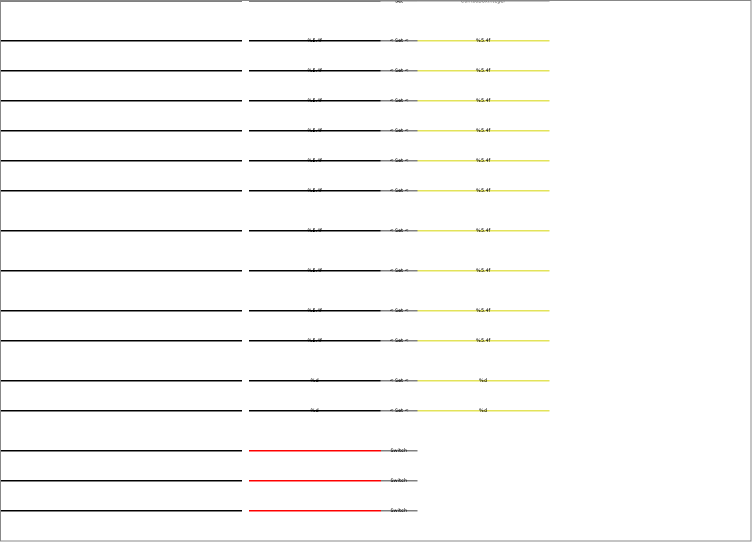
VISUALIZATION Visu_Mparam_Heat  // 752x542
    Frame (0,40 750x30)
        shows Param_LREAL(nIdx := 4)
    Frame (0,70 750x30)
        shows Param_LREAL(nIdx := 6)
    Frame (0,100 750x30)
        shows Param_LREAL(nIdx := 8)
    Frame (0,130 750x30)
        shows Param_LREAL(nIdx := 10)
    Frame (0,380 750x30)
        shows Param_DINT(nIdx := 11)
    Frame (0,0 750x30)
        shows Param_ENUM_SelOut(nIdx := GlobalOne)
    Frame (0,160 750x30)
        shows Param_LREAL(nIdx := 16)
    Frame (0,190 750x30)
        shows Param_LREAL(nIdx := 17)
    Frame (0,230 750x30)
        shows Param_LREAL(nIdx := 21)
    Frame (0,310 750x30)
        shows Param_LREAL(nIdx := 37)
    Frame (0,340 750x30)
        shows Param_LREAL(nIdx := 38)
    Frame (0,450 750x30)
        shows Param_BOOL(nIdx := GlobalOne)
    Frame (0,480 750x30)
        shows Param_BOOL(nIdx := 3)
    Frame (0,510 750x30)
        shows Param_BOOL(nIdx := 18)
    Frame (0,270 750x30)
        shows Param_LREAL(nIdx := 32)
    Frame (0,410 750x30)
        shows Param_DINT(nIdx := 12)
END_VISUALIZATION

// ---- VISUs/Pages/Machine/Subpage/Visu_Mparam_Supply.TcVIS
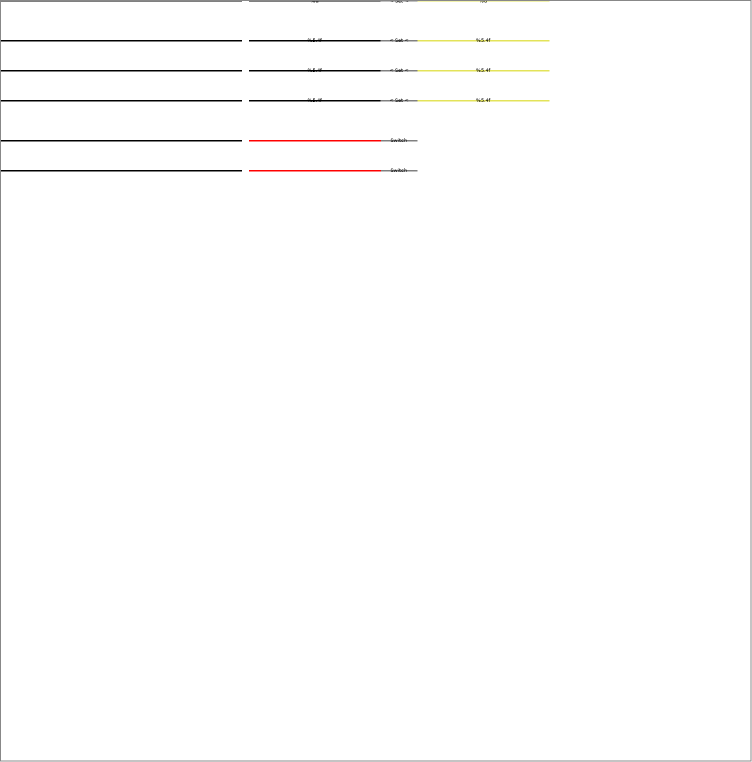
VISUALIZATION Visu_Mparam_Supply  // 752x762
    Frame (0,40 750x30)
        shows Param_LREAL(nIdx := 21)
    Frame (0,70 750x30)
        shows Param_LREAL(nIdx := 22)
    Frame (0,100 750x30)
        shows Param_LREAL(nIdx := 23)
    Frame (0,0 750x30)
        shows Param_DINT(nIdx := 6)
    Frame (0,140 750x30)
        shows Param_BOOL(nIdx := 11)
    Frame (0,170 750x30)
        shows Param_BOOL(nIdx := 15)
    Rectangle (0,730 750x30)
END_VISUALIZATION

// ---- VISUs/Pages/Machine/Subpage/Visu_Mparam_Temperatur.TcVIS
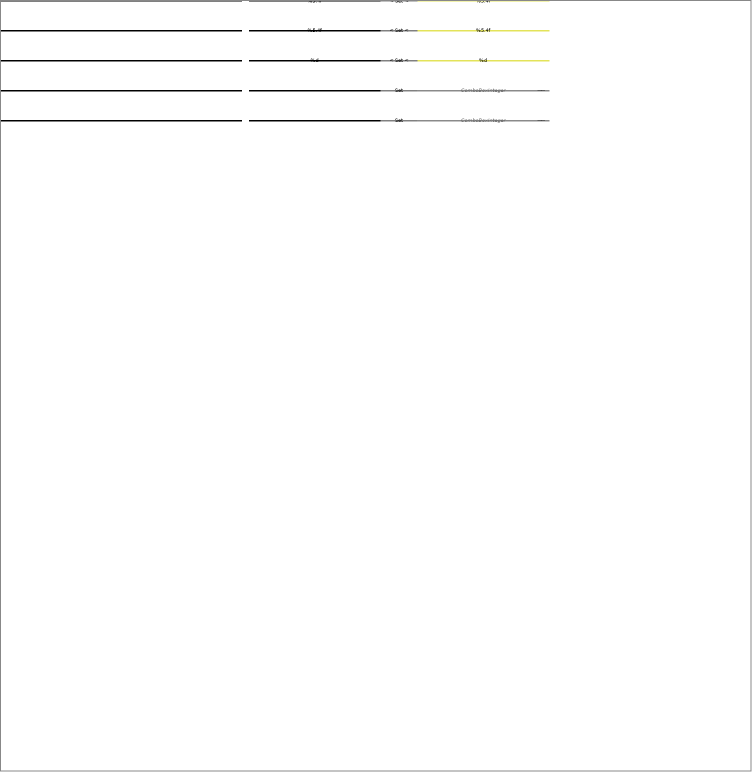
VISUALIZATION Visu_Mparam_Temperatur  // 752x772
    Frame (0,0 750x30)
        shows Param_LREAL(nIdx := GlobalOne)
    Frame (0,30 750x30)
        shows Param_LREAL(nIdx := 2)
    Frame (0,60 750x30)
        shows Param_DINT(nIdx := 9)
    Frame (0,90 750x30)
        shows Param_ENUM_TermType(nIdx := 3)
    Frame (0,120 750x30)
        shows Param_ENUM_SensType(nIdx := 4)
    Rectangle (0,740 750x30)
END_VISUALIZATION

// ---- VISUs/Pages/Machine/Visu_MParam.TcVIS
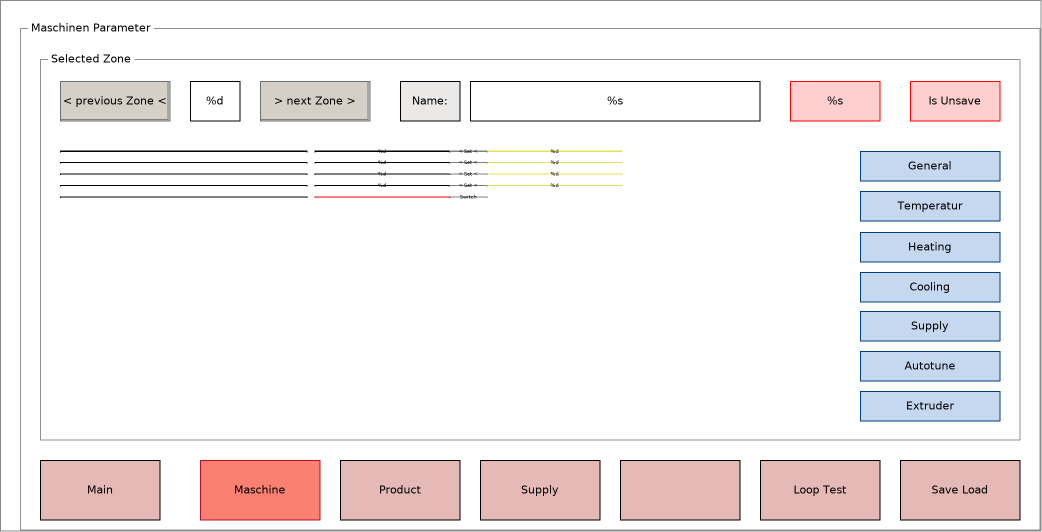
VISUALIZATION Visu_MParam  // 1042x532
    GroupBox (20,20 1020x510), "Maschinen Parameter"
        Rectangle (20,440 120x60), "Main"
            OnMouseClick: change screen: Visu_Main
        Rectangle (880,440 120x60), "Save Load"
            OnMouseClick: change screen: Visu_SaveLoad
        Rectangle (320,440 120x60), "Product"
            OnMouseClick: change screen: Visu_PParam
        Rectangle (180,440 120x60), "Maschine"
            OnMouseClick: change screen: Visu_MParam
        Rectangle (460,440 120x60), "Supply"
            OnMouseClick: change screen: Visu_Supply
        Rectangle (600,440 120x60)
        GroupBox (20,31 980x389), "Selected Zone"
            Rectangle (150,30 50x40), "%d", text variable: nVisuCount
            Button (20,30 110x40), "< previous Zone <"
                tap bVisuBefore
            Button (220,30 110x40), "> next Zone >"
                tap bVisuNext
            Rectangle (750,30 90x40), "%s", text variable: stMParam_Visu.sInUse, colour toggle: aaaPfwTempMparamFromHmi[nVisuCount].InUse
                OnMouseClick: toggle aaaPfwTempMparamFromHmi[nVisuCount].InUse
                OnMouseClick: execute { stParamsUnsave.mParams[nVisuCount]:=TRUE; }
            Rectangle (430,30 290x40), "%s", text variable: aaaPfwTempMparamFromHmi[nVisuCount].ZoneName
                OnMouseClick: write the text variable via Edit
                OnMouseClick: execute { stParamsUnsave.mParams[nVisuCount]:=TRUE; }
            Rectangle (360,30 60x40), "Name:"
            Rectangle (870,30 90x40), "Is Unsave", invisible if: Not stParamsUnsave.mParams[nVisuCount]
                OnMouseClick: execute { aaaPfwTempMparamFromHmi[nVisuCount].SaveDelay:=1000; stParamsUnsave.mParams[nVisuCount]:=FALSE; }
            Rectangle (820,100 140x30), "General", colour toggle: stMParam_Visu.nActiveParamList=0
                OnMouseClick: execute { stMParam_Visu.nActiveParamList:=0; }
            Frame (20,100 790x280), frame switch variable: stMParam_Visu.nActiveParamList
                shows Visu_Mparam_General()
                shows Visu_Mparam_Temperatur()
                shows Visu_Mparam_Heat()
                shows Visu_Mparam_Cool()
                shows Visu_Mparam_Supply()
                shows Visu_Mparam_Autotune()
                shows Visu_Mparam_Extruder()
            Rectangle (820,221 140x30), "Cooling", colour toggle: stMParam_Visu.nActiveParamList=3
                OnMouseClick: execute { stMParam_Visu.nActiveParamList:=3; }
            Rectangle (820,181 140x30), "Heating", colour toggle: stMParam_Visu.nActiveParamList=2
                OnMouseClick: execute { stMParam_Visu.nActiveParamList:=2; }
            Rectangle (820,340 140x30), "Extruder", colour toggle: stMParam_Visu.nActiveParamList=6
                OnMouseClick: execute { stMParam_Visu.nActiveParamList:=6; }
            Rectangle (820,300 140x30), "Autotune", colour toggle: stMParam_Visu.nActiveParamList=5
                OnMouseClick: execute { stMParam_Visu.nActiveParamList:=5; }
            Rectangle (820,260 140x30), "Supply", colour toggle: stMParam_Visu.nActiveParamList=4
                OnMouseClick: execute { stMParam_Visu.nActiveParamList:=4; }
            Rectangle (820,140 140x30), "Temperatur", colour toggle: stMParam_Visu.nActiveParamList=1
                OnMouseClick: execute { stMParam_Visu.nActiveParamList:=1; }
        Rectangle (740,440 120x60), "Loop Test"
            OnMouseClick: change screen: Visu_LoopTest
END_VISUALIZATION

// ---- VISUs/Pages/Product/Param_LREAL_Pparam.TcVIS
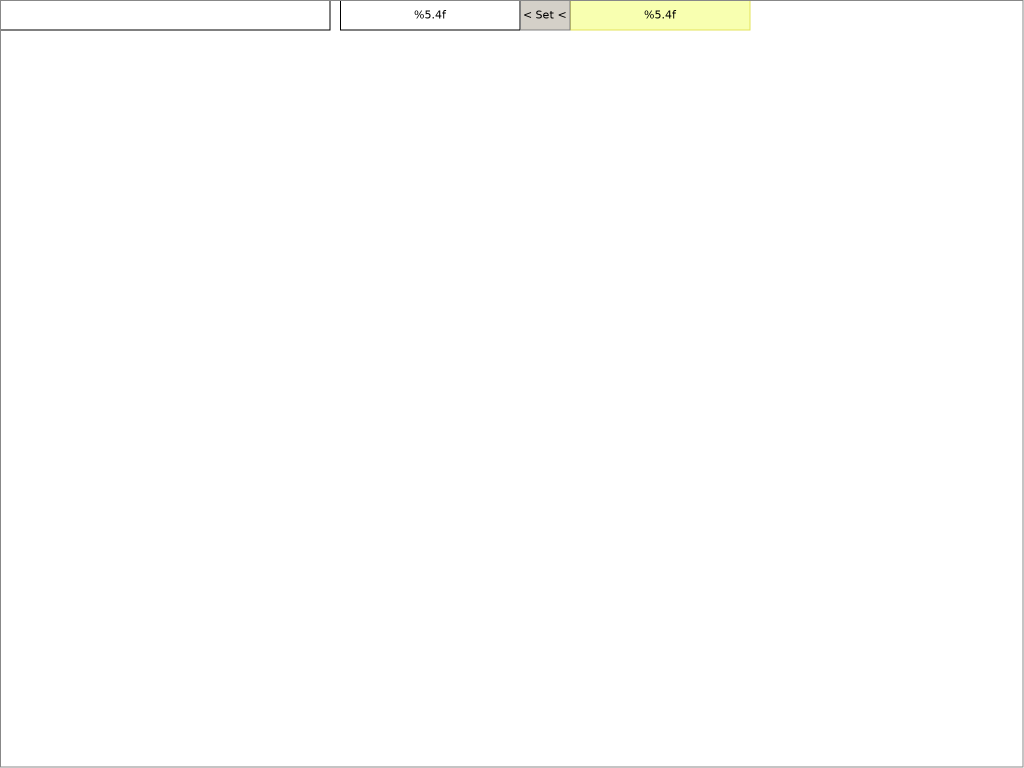
VISUALIZATION Param_LREAL_Pparam  // 1024x768
VAR_INPUT
	nIdx:		INT;
END_VAR
    Rectangle (340,0 180x30), "%5.4f", text variable: stPParam_Visu.fLrealAktValue[nIdx]
    Rectangle (0,0 330x30), text list: 'TL_Pparmas', text index: nIdx
    Rectangle (570,0 180x30), "%5.4f", text variable: stPParam_Visu.fLrealNewValue[nIdx]
        OnMouseClick: write the text variable via Default
    Rectangle (520,0 50x30), "< Set <"
        OnMouseClick: execute { stPParam_Visu.bLrealSetValue[nIdx]:=TRUE; }
END_VISUALIZATION

// ---- VISUs/Pages/Product/Visu_PParam.TcVIS
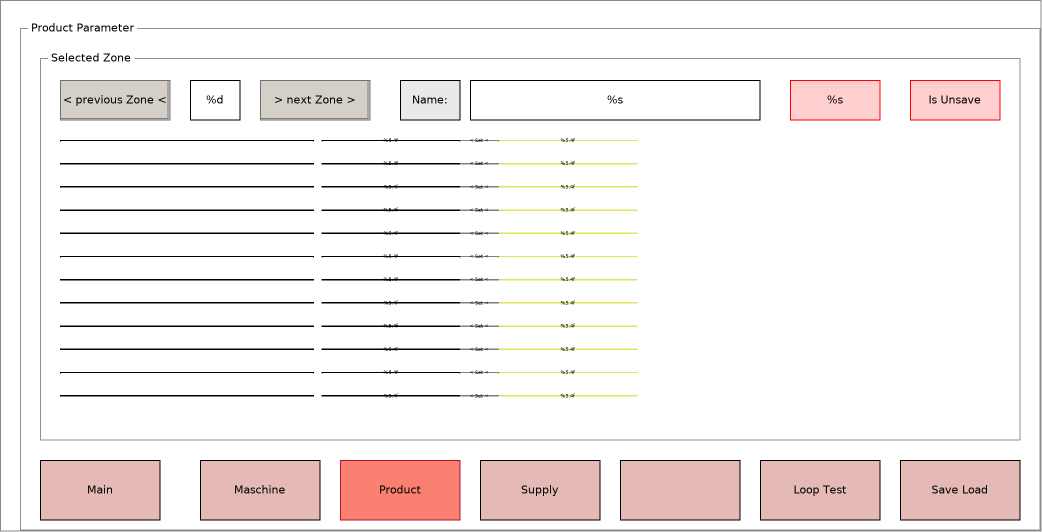
VISUALIZATION Visu_PParam  // 1042x532
    GroupBox (20,20 1020x510), "Product Parameter"
        Rectangle (20,440 120x60), "Main"
            OnMouseClick: change screen: Visu_Main
        Rectangle (880,440 120x60), "Save Load"
            OnMouseClick: change screen: Visu_SaveLoad
        Rectangle (320,440 120x60), "Product"
            OnMouseClick: change screen: Visu_PParam
        GroupBox (20,30 980x390), "Selected Zone"
            Rectangle (150,30 50x40), "%d", text variable: nVisuCount
            Button (20,30 110x40), "< previous Zone <"
                tap bVisuBefore
            Button (220,30 110x40), "> next Zone >"
                tap bVisuNext
            Rectangle (430,30 290x40), "%s", text variable: aaaPfwTempMparamFromHmi[nVisuCount].ZoneName
            Rectangle (360,30 60x40), "Name:"
            Frame (20,90 790x280)
                shows Visu_PParam_Params()
                shows Visu_MParam_ENUM()
                shows Visu_MParam_BOOL()
                shows Visu_MParam_INT()
            Rectangle (870,30 90x40), "Is Unsave", invisible if: Not stParamsUnsave.pParams[nVisuCount]
                OnMouseClick: execute { aaaPfwTempPparamFromHmi[nVisuCount].SaveDelay:=1000; stParamsUnsave.pParams[nVisuCount]:=FALSE; }
        Rectangle (180,440 120x60), "Maschine"
            OnMouseClick: change screen: Visu_MParam
    Rectangle (480,460 120x60), "Supply"
        OnMouseClick: change screen: Visu_Supply
    Rectangle (620,460 120x60)
    Rectangle (760,460 120x60), "Loop Test"
        OnMouseClick: change screen: Visu_LoopTest
    Rectangle (790,80 90x40), "%s", text variable: stMParam_Visu.sInUse, colour toggle: aaaPfwTempMparamFromHmi[nVisuCount].InUse
        OnMouseClick: toggle aaaPfwTempMparamFromHmi[nVisuCount].InUse
        OnMouseClick: execute { stParamsUnsave.mParams[nVisuCount]:=TRUE; }
END_VISUALIZATION

// ---- VISUs/Pages/Product/Visu_PParam_Params.TcVIS
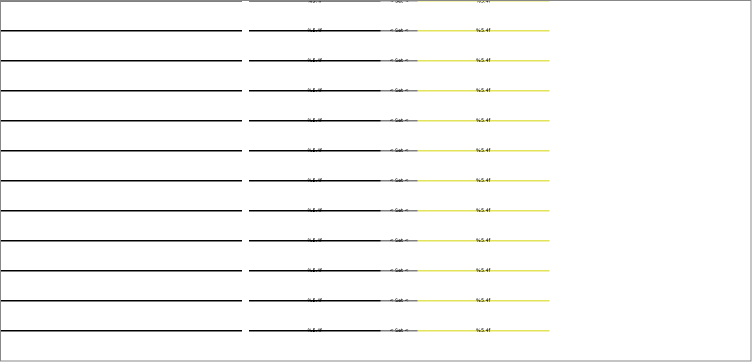
VISUALIZATION Visu_PParam_Params  // 752x362
    Frame (0,0 750x30)
        shows Param_LREAL_Pparam(nIdx := GlobalOne)
    Frame (0,30 750x30)
        shows Param_LREAL_Pparam(nIdx := 2)
    Frame (0,60 750x30)
        shows Param_LREAL_Pparam(nIdx := 3)
    Frame (0,90 750x30)
        shows Param_LREAL_Pparam(nIdx := 4)
    Frame (0,120 750x30)
        shows Param_LREAL_Pparam(nIdx := 5)
    Frame (0,150 750x30)
        shows Param_LREAL_Pparam(nIdx := 6)
    Frame (0,180 750x30)
        shows Param_LREAL_Pparam(nIdx := 7)
    Frame (0,210 750x30)
        shows Param_LREAL_Pparam(nIdx := 8)
    Frame (0,240 750x30)
        shows Param_LREAL_Pparam(nIdx := 9)
    Frame (0,270 750x30)
        shows Param_LREAL_Pparam(nIdx := 10)
    Frame (0,300 750x30)
        shows Param_LREAL_Pparam(nIdx := 11)
    Frame (0,330 750x30)
        shows Param_LREAL_Pparam(nIdx := 12)
END_VISUALIZATION

// ---- VISUs/Pages/Supply/Param_LREAL_Supply.TcVIS
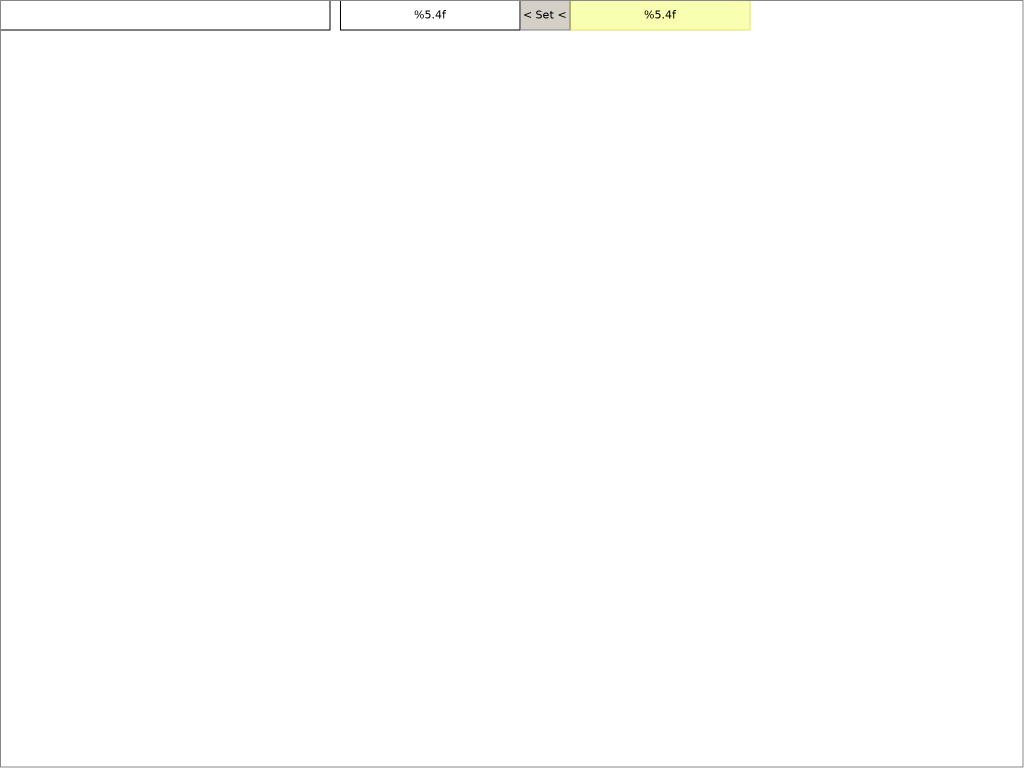
VISUALIZATION Param_LREAL_Supply  // 1024x768
VAR_INPUT
	nIdx:		INT;
END_VAR
    Rectangle (340,0 180x30), "%5.4f", text variable: stSupply_Visu.fLrealAktValue[nIdx]
    Rectangle (0,0 330x30), text list: 'TL_Supply', text index: nIdx
    Rectangle (570,0 180x30), "%5.4f", text variable: stSupply_Visu.fLrealNewValue[nIdx]
        OnMouseClick: write the text variable via Default
    Rectangle (520,0 50x30), "< Set <"
        OnMouseClick: execute { stSupply_Visu.bLrealSetValue[nIdx]:=TRUE; }
END_VISUALIZATION

// ---- VISUs/Pages/Supply/Visu_Supply.TcVIS
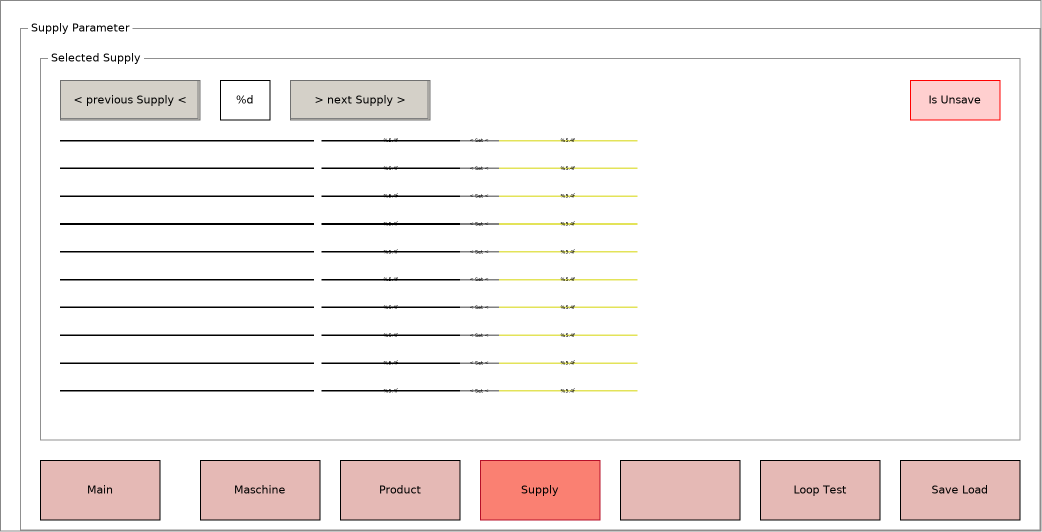
VISUALIZATION Visu_Supply  // 1042x532
    GroupBox (20,20 1020x510), "Supply Parameter"
        Rectangle (20,440 120x60), "Main"
            OnMouseClick: change screen: Visu_Main
        Rectangle (880,440 120x60), "Save Load"
            OnMouseClick: change screen: Visu_SaveLoad
        Rectangle (320,440 120x60), "Product"
            OnMouseClick: change screen: Visu_PParam
        Rectangle (180,440 120x60), "Maschine"
            OnMouseClick: change screen: Visu_MParam
        Rectangle (460,440 120x60), "Supply"
            OnMouseClick: change screen: Visu_Supply
        Rectangle (600,440 120x60)
        Rectangle (740,440 120x60), "Loop Test"
            OnMouseClick: change screen: Visu_LoopTest
        GroupBox (20,30 980x390), "Selected Supply"
            Rectangle (180,30 50x40), "%d", text variable: nSupplyCnt
            Button (20,30 140x40), "< previous Supply <"
                OnMouseClick: execute { nSupplyCnt:= MAX(cnPfwAppSupplyFirst, nSupplyCnt-1); }
            Button (250,30 140x40), "> next Supply >"
                OnMouseClick: execute { nSupplyCnt:= MIN(cnPfwAppSupplyLast, nSupplyCnt+1); }
            Rectangle (870,30 90x40), "Is Unsave", invisible if: Not stParamsUnsave.supply[nSupplyCnt]
                OnMouseClick: execute { stPfwSupplyLineCfg[nSupplyCnt].SaveDelay:=1000; stParamsUnsave.supply[nSupplyCnt]:=FALSE; }
            Frame (20,90 790x280)
                shows Visu_Supply_Params()
                shows Visu_MParam_ENUM()
                shows Visu_MParam_BOOL()
                shows Visu_MParam_INT()
END_VISUALIZATION

// ---- VISUs/Pages/Supply/Visu_Supply_Params.TcVIS
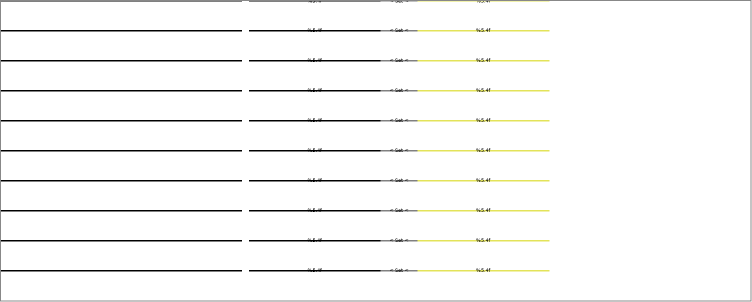
VISUALIZATION Visu_Supply_Params  // 752x302
    Frame (0,0 750x30)
        shows Param_LREAL_Supply(nIdx := GlobalOne)
    Frame (0,30 750x30)
        shows Param_LREAL_Supply(nIdx := 2)
    Frame (0,60 750x30)
        shows Param_LREAL_Supply(nIdx := 3)
    Frame (0,120 750x30)
        shows Param_LREAL_Supply(nIdx := 5)
    Frame (0,90 750x30)
        shows Param_LREAL_Supply(nIdx := 4)
    Frame (0,270 750x30)
        shows Param_LREAL_Supply(nIdx := 10)
    Frame (0,240 750x30)
        shows Param_LREAL_Supply(nIdx := 9)
    Frame (0,210 750x30)
        shows Param_LREAL_Supply(nIdx := 8)
    Frame (0,180 750x30)
        shows Param_LREAL_Supply(nIdx := 7)
    Frame (0,150 750x30)
        shows Param_LREAL_Supply(nIdx := 6)
END_VISUALIZATION

// ---- VISUs/Pages/Visu_Main.TcVIS
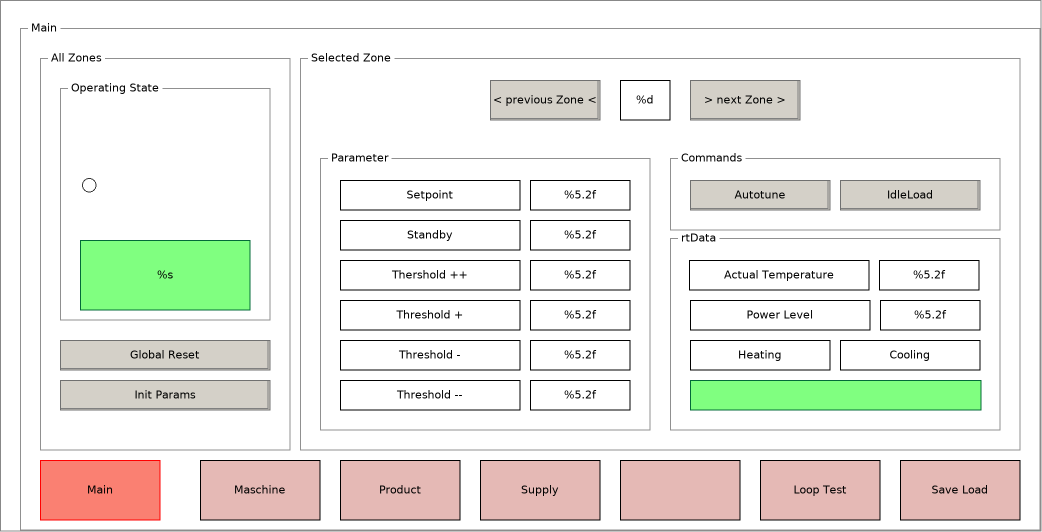
VISUALIZATION Visu_Main  // 1042x532
    GroupBox (20,20 1020x510), "Main"
        Rectangle (20,440 120x60), "Main"
            OnMouseClick: change screen: Visu_Main
        Rectangle (880,440 120x60), "Save Load"
            OnMouseClick: change screen: Visu_SaveLoad
        Rectangle (320,440 120x60), "Product"
            OnMouseClick: change screen: Visu_PParam
        Rectangle (180,440 120x60), "Maschine"
            OnMouseClick: change screen: Visu_MParam
    GroupBox (40,50 250x400), "All Zones", input disabled if: MAIN.eState<>eMainSM_Idle
        GroupBox (20,30 210x240), "Operating State", input disabled if: MAIN.eState<>eMainSM_Idle
            RadioButton (20,30 150x150), variable: eStatus
                Areas[0]: Text=Off
                Areas[1]: Text=Standby
                Areas[2]: Text=On
                Areas[3]: Text=Autotune
                Areas[4]: Text=Idle Load
            Rectangle (20,160 170x70), "%s", text variable: sErrorText, colour toggle: bGlobalError
        Button (20,330 210x30), "Init Params"
            tap bParamsInit
        Button (20,290 210x30), "Global Reset"
            tap aaaTempFault_Reset
    GroupBox (300,50 720x400), "Selected Zone"
        Rectangle (320,30 50x40), "%d", text variable: nVisuCount
        Button (190,30 110x40), "< previous Zone <"
            tap bVisuBefore
        Button (390,30 110x40), "> next Zone >"
            tap bVisuNext
        GroupBox (20,100 330x280), "Parameter"
            Rectangle (20,30 180x30), "Setpoint"
            Rectangle (20,70 180x30), "Standby"
            Rectangle (20,110 180x30), "Thershold ++"
            Rectangle (20,150 180x30), "Threshold +"
            Rectangle (20,190 180x30), "Threshold -"
            Rectangle (20,230 180x30), "Threshold --"
            Rectangle (210,30 100x30), "%5.2f", text variable: aaaPfwTempPparamFromHmi[nVisuCount].Setpoint
            Rectangle (210,70 100x30), "%5.2f", text variable: aaaPfwTempPparamFromHmi[nVisuCount].StandbySetpoint
            Rectangle (210,110 100x30), "%5.2f", text variable: aaaPfwTempPparamFromHmi[nVisuCount].Threshold_PP
            Rectangle (210,150 100x30), "%5.2f", text variable: aaaPfwTempPparamFromHmi[nVisuCount].Threshold_P
            Rectangle (210,190 100x30), "%5.2f", text variable: aaaPfwTempPparamFromHmi[nVisuCount].Threshold_M
            Rectangle (210,230 100x30), "%5.2f", text variable: aaaPfwTempPparamFromHmi[nVisuCount].Threshold_MM
        GroupBox (370,180 330x200), "rtData"
            Rectangle (210,70 100x30), "%5.2f", text variable: aaaPfwTempToHmi[nVisuCount].PowerLevel
            Rectangle (19,30 180x30), "Actual Temperature"
            Rectangle (209,30 100x30), "%5.2f", text variable: aaaPfwTempToHmi[nVisuCount].ActualTemp
            Rectangle (20,70 180x30), "Power Level"
            Rectangle (170,110 140x30), "Cooling", colour toggle: aaaPfwTempToHmi[nVisuCount].Cooling
            Rectangle (20,110 140x30), "Heating", colour toggle: aaaPfwTempToHmi[nVisuCount].Heating
            Rectangle (20,150 291x30), colour toggle: aaaPfwTempToHmi[nVisuCount].Error, text list: 'TL_TcPfw_ErrorId', text index: INT_TO_STRING(aaaPfwTempToHmi[nVisuCount].ErrorId)
                OnMouseClick: ChangeLanguage ChangeLanguage=en
        GroupBox (370,100 330x80), "Commands", input disabled if: aaaPfwTempMparamFromHmi[nVisuCount].Autotune OR aaaPfwTempMparamFromHmi[nVisuCount].Ena_TuneIdleLoad OR MAIN.eState<>eMainSM_Idle
            Button (20,30 140x30), "Autotune"
                tap bVisuAutotune
            Button (170,30 140x30), "IdleLoad"
                tap bVisuIdleLoad
    Rectangle (480,460 120x60), "Supply"
        OnMouseClick: change screen: Visu_Supply
    Rectangle (620,460 120x60)
    Rectangle (760,460 120x60), "Loop Test"
        OnMouseClick: change screen: Visu_LoopTest
END_VISUALIZATION
